    movel([0.108548, -1.229581, -2.664379, -0.818429, 1.570796, 1.679344],accel_mss,speed_ms,0,blend_radius_m)
    movel([0.107464, -1.232991, -2.662638, -0.816759, 1.570796, 1.678260],accel_mss,speed_ms,0,blend_radius_m)
    movel([0.106659, -1.236345, -2.660913, -0.815131, 1.570796, 1.677455],accel_mss,speed_ms,0,blend_radius_m)
    movel([0.106148, -1.239625, -2.659213, -0.813551, 1.570796, 1.676944],accel_mss,speed_ms,0,blend_radius_m)
    movel([0.105928, -1.242820, -2.657545, -0.812024, 1.570796, 1.676724],accel_mss,speed_ms,0,blend_radius_m)
    movel([0.106013, -1.245914, -2.655918, -0.810557, 1.570796, 1.676809],accel_mss,speed_ms,0,blend_radius_m)
    movel([0.106368, -1.248628, -2.654481, -0.809280, 1.570796, 1.677165],accel_mss,speed_ms,0,blend_radius_m)
    movel([0.106979, -1.251120, -2.653154, -0.808115, 1.570796, 1.677775],accel_mss,speed_ms,0,blend_radius_m)
    movel([0.107817, -1.253397, -2.651935, -0.807057, 1.570796, 1.678614],accel_mss,speed_ms,0,blend_radius_m)
    movel([0.108863, -1.255463, -2.650824, -0.806102, 1.570796, 1.679659],accel_mss,speed_ms,0,blend_radius_m)
    movel([0.110091, -1.257325, -2.649818, -0.805246, 1.570796, 1.680887],accel_mss,speed_ms,0,blend_radius_m)
    movel([0.111476, -1.258987, -2.648916, -0.804485, 1.570796, 1.682272],accel_mss,speed_ms,0,blend_radius_m)
    movel([0.112995, -1.260456, -2.648117, -0.803816, 1.570796, 1.683792],accel_mss,speed_ms,0,blend_radius_m)
    movel([0.114629, -1.261734, -2.647419, -0.803236, 1.570796, 1.685426],accel_mss,speed_ms,0,blend_radius_m)
    movel([0.116356, -1.262825, -2.646822, -0.802742, 1.570796, 1.687152],accel_mss,speed_ms,0,blend_radius_m)
    movel([0.118150, -1.263736, -2.646322, -0.802331, 1.570796, 1.688947],accel_mss,speed_ms,0,blend_radius_m)
    movel([0.119994, -1.264467, -2.645920, -0.802002, 1.570796, 1.690791],accel_mss,speed_ms,0,blend_radius_m)
    movel([0.121863, -1.265023, -2.645614, -0.801752, 1.570796, 1.692659],accel_mss,speed_ms,0,blend_radius_m)
    movel([0.123738, -1.265404, -2.645404, -0.801581, 1.570796, 1.694534],accel_mss,speed_ms,0,blend_radius_m)
    movel([0.125599, -1.265611, -2.645290, -0.801488, 1.570796, 1.696395],accel_mss,speed_ms,0,blend_radius_m)
    movel([0.127421, -1.265653, -2.645267, -0.801469, 1.570796, 1.698217],accel_mss,speed_ms,0,blend_radius_m)
    movel([0.129187, -1.265524, -2.645338, -0.801527, 1.570796, 1.699983],accel_mss,speed_ms,0,blend_radius_m)
    movel([0.130799, -1.262042, -2.647250, -0.803096, 1.570796, 1.701596],accel_mss,speed_ms,0,blend_radius_m)
    movel([0.127034, -1.261584, -2.647501, -0.803304, 1.570796, 1.697831],accel_mss,speed_ms,0,blend_radius_m)
    movel([0.123670, -1.260748, -2.647958, -0.803684, 1.570796, 1.694467],accel_mss,speed_ms,0,blend_radius_m)
    movel([0.120699, -1.259562, -2.648603, -0.804223, 1.570796, 1.691495],accel_mss,speed_ms,0,blend_radius_m)
    movel([0.118110, -1.258051, -2.649424, -0.804913, 1.570796, 1.688906],accel_mss,speed_ms,0,blend_radius_m)
    movel([0.115901, -1.256233, -2.650408, -0.805748, 1.570796, 1.686697],accel_mss,speed_ms,0,blend_radius_m)
    movel([0.114064, -1.254135, -2.651539, -0.806715, 1.570796, 1.684861],accel_mss,speed_ms,0,blend_radius_m)
    movel([0.112599, -1.251775, -2.652804, -0.807810, 1.570796, 1.683395],accel_mss,speed_ms,0,blend_radius_m)
    movel([0.111497, -1.249180, -2.654188, -0.809021, 1.570796, 1.682294],accel_mss,speed_ms,0,blend_radius_m)
    movel([0.110757, -1.246371, -2.655676, -0.810342, 1.570796, 1.681553],accel_mss,speed_ms,0,blend_radius_m)
    movel([0.110373, -1.243371, -2.657256, -0.811762, 1.570796, 1.681169],accel_mss,speed_ms,0,blend_radius_m)
    movel([0.110346, -1.240205, -2.658911, -0.813273, 1.570796, 1.681143],accel_mss,speed_ms,0,blend_radius_m)
    movel([0.110668, -1.236899, -2.660627, -0.814863, 1.570796, 1.681464],accel_mss,speed_ms,0,blend_radius_m)
    movel([0.111341, -1.233474, -2.662391, -0.816524, 1.570796, 1.682137],accel_mss,speed_ms,0,blend_radius_m)
    movel([0.112362, -1.229961, -2.664186, -0.818242, 1.570796, 1.683158],accel_mss,speed_ms,0,blend_radius_m)
    movel([0.113724, -1.226382, -2.666000, -0.820007, 1.570796, 1.684520],accel_mss,speed_ms,0,blend_radius_m)
    movel([0.115426, -1.222769, -2.667817, -0.821803, 1.570796, 1.686223],accel_mss,speed_ms,0,blend_radius_m)
    movel([0.117544, -1.218987, -2.669702, -0.823699, 1.570796, 1.688341],accel_mss,speed_ms,0,blend_radius_m)
    movel([0.119932, -1.215305, -2.671523, -0.825562, 1.570796, 1.690729],accel_mss,speed_ms,0,blend_radius_m)
    movel([0.122570, -1.211733, -2.673273, -0.827383, 1.570796, 1.693366],accel_mss,speed_ms,0,blend_radius_m)
    movel([0.125434, -1.208299, -2.674943, -0.829147, 1.570796, 1.696231],accel_mss,speed_ms,0,blend_radius_m)
    movel([0.128500, -1.205022, -2.676524, -0.830843, 1.570796, 1.699296],accel_mss,speed_ms,0,blend_radius_m)
    movel([0.131747, -1.201919, -2.678010, -0.832459, 1.570796, 1.702544],accel_mss,speed_ms,0,blend_radius_m)
    movel([0.135148, -1.199015, -2.679392, -0.833982, 1.570796, 1.705945],accel_mss,speed_ms,0,blend_radius_m)
    movel([0.138679, -1.196328, -2.680662, -0.835399, 1.570796, 1.709475],accel_mss,speed_ms,0,blend_radius_m)
    movel([0.142314, -1.193882, -2.681811, -0.836696, 1.570796, 1.713110],accel_mss,speed_ms,0,blend_radius_m)
    movel([0.146026, -1.191698, -2.682831, -0.837859, 1.570796, 1.716822],accel_mss,speed_ms,0,blend_radius_m)
    movel([0.149789, -1.189798, -2.683715, -0.838876, 1.570796, 1.720586],accel_mss,speed_ms,0,blend_radius_m)
    movel([0.153576, -1.188205, -2.684453, -0.839731, 1.570796, 1.724373],accel_mss,speed_ms,0,blend_radius_m)
    movel([0.157357, -1.186934, -2.685039, -0.840415, 1.570796, 1.728154],accel_mss,speed_ms,0,blend_radius_m)
    movel([0.161105, -1.186010, -2.685465, -0.840914, 1.570796, 1.731901],accel_mss,speed_ms,0,blend_radius_m)
    movel([0.164790, -1.185454, -2.685721, -0.841214, 1.570796, 1.735586],accel_mss,speed_ms,0,blend_radius_m)
    movel([0.168388, -1.185281, -2.685800, -0.841308, 1.570796, 1.739184],accel_mss,speed_ms,0,blend_radius_m)
    movel([0.171744, -1.185486, -2.685706, -0.841197, 1.570796, 1.742541],accel_mss,speed_ms,0,blend_radius_m)
    movel([0.174813, -1.186046, -2.685449, -0.840895, 1.570796, 1.745609],accel_mss,speed_ms,0,blend_radius_m)
    movel([0.177595, -1.186957, -2.685029, -0.840403, 1.570796, 1.748391],accel_mss,speed_ms,0,blend_radius_m)
    movel([0.180079, -1.188212, -2.684450, -0.839728, 1.570796, 1.750875],accel_mss,speed_ms,0,blend_radius_m)
    movel([0.182267, -1.189808, -2.683710, -0.838870, 1.570796, 1.753063],accel_mss,speed_ms,0,blend_radius_m)
    movel([0.184151, -1.191740, -2.682812, -0.837837, 1.570796, 1.754947],accel_mss,speed_ms,0,blend_radius_m)
    movel([0.185731, -1.194002, -2.681755, -0.836632, 1.570796, 1.756527],accel_mss,speed_ms,0,blend_radius_m)
    movel([0.187008, -1.196584, -2.680541, -0.835264, 1.570796, 1.757804],accel_mss,speed_ms,0,blend_radius_m)
    movel([0.188195, -1.200365, -2.678751, -0.833273, 1.570796, 1.758991],accel_mss,speed_ms,0,blend_radius_m)
    movel([0.188551, -1.202327, -2.677816, -0.832246, 1.570796, 1.759347],accel_mss,speed_ms,0,blend_radius_m)
    movel([0.188803, -1.206387, -2.675867, -0.830135, 1.570796, 1.759599],accel_mss,speed_ms,0,blend_radius_m)
    movel([0.188703, -1.208484, -2.674853, -0.829051, 1.570796, 1.759500],accel_mss,speed_ms,0,blend_radius_m)
    movel([0.188070, -1.212794, -2.672754, -0.826840, 1.570796, 1.758866],accel_mss,speed_ms,0,blend_radius_m)
    movel([0.187544, -1.215004, -2.671670, -0.825715, 1.570796, 1.758341],accel_mss,speed_ms,0,blend_radius_m)
    movel([0.186076, -1.219536, -2.669430, -0.823423, 1.570796, 1.756872],accel_mss,speed_ms,0,blend_radius_m)
    movel([0.185142, -1.221849, -2.668277, -0.822263, 1.570796, 1.755939],accel_mss,speed_ms,0,blend_radius_m)
    movel([0.182886, -1.226576, -2.665902, -0.819911, 1.570796, 1.753682],accel_mss,speed_ms,0,blend_radius_m)
    movel([0.180136, -1.231422, -2.663441, -0.817526, 1.570796, 1.750932],accel_mss,speed_ms,0,blend_radius_m)
    movel([0.183278, -1.232244, -2.663021, -0.817124, 1.570796, 1.754074],accel_mss,speed_ms,0,blend_radius_m)
    movel([0.185050, -1.229577, -2.664381, -0.818430, 1.570796, 1.755846],accel_mss,speed_ms,0,blend_radius_m)
    movel([0.185168, -1.229377, -2.664483, -0.818529, 1.570796, 1.755964],accel_mss,speed_ms,0,blend_radius_m)
    speed_ms = 0.005
    # Splitting Linear movement in 4 (instruction 1141: MoveL 1073)
    movel([0.185168, -1.226955, -2.663319, -0.822115, 1.570796, 1.755964],accel_mss,speed_ms,0,blend_radius_m)
    movel([0.185168, -1.224548, -2.662151, -0.825690, 1.570796, 1.755964],accel_mss,speed_ms,0,blend_radius_m)
    movel([0.185168, -1.222156, -2.660979, -0.829253, 1.570796, 1.755964],accel_mss,speed_ms,0,blend_radius_m)
    movel([0.185168, -1.219779, -2.659804, -0.832806, 1.570796, 1.755964],accel_mss,speed_ms,0,blend_radius_m)
    speed_ms = 0.040
    # Splitting Linear movement in 8 (instruction 1143: MoveL 1074)
    movel([0.184772, -1.222069, -2.658652, -0.831667, 1.570796, 1.755568],accel_mss,speed_ms,0,blend_radius_m)
    movel([0.184379, -1.224351, -2.657499, -0.830539, 1.570796, 1.755175],accel_mss,speed_ms,0,blend_radius_m)
    movel([0.183987, -1.226625, -2.656343, -0.829421, 1.570796, 1.754783],accel_mss,speed_ms,0,blend_radius_m)
    movel([0.183597, -1.228891, -2.655186, -0.828312, 1.570796, 1.754394],accel_mss,speed_ms,0,blend_radius_m)
    movel([0.183210, -1.231149, -2.654027, -0.827213, 1.570796, 1.754006],accel_mss,speed_ms,0,blend_radius_m)
    movel([0.182824, -1.233399, -2.652866, -0.826124, 1.570796, 1.753620],accel_mss,speed_ms,0,blend_radius_m)
    movel([0.182440, -1.235641, -2.651703, -0.825045, 1.570796, 1.753237],accel_mss,speed_ms,0,blend_radius_m)
    movel([0.182059, -1.237876, -2.650538, -0.823975, 1.570796, 1.752855],accel_mss,speed_ms,0,blend_radius_m)
    speed_ms = 0.005
    # Splitting Linear movement in 4 (instruction 1145: MoveL 1075)
    movel([0.182059, -1.240234, -2.651693, -0.820462, 1.570796, 1.752855],accel_mss,speed_ms,0,blend_radius_m)
    movel([0.182059, -1.242607, -2.652844, -0.816938, 1.570796, 1.752855],accel_mss,speed_ms,0,blend_radius_m)
    movel([0.182059, -1.244994, -2.653991, -0.813404, 1.570796, 1.752855],accel_mss,speed_ms,0,blend_radius_m)
    movel([0.182059, -1.247395, -2.655135, -0.809860, 1.570796, 1.752855],accel_mss,speed_ms,0,blend_radius_m)
    speed_ms = 0.035
    movel([0.183122, -1.249001, -2.654283, -0.809105, 1.570796, 1.753919],accel_mss,speed_ms,0,blend_radius_m)
    movel([0.184641, -1.250273, -2.653606, -0.808510, 1.570796, 1.755437],accel_mss,speed_ms,0,blend_radius_m)
    movel([0.186541, -1.251208, -2.653107, -0.808074, 1.570796, 1.757337],accel_mss,speed_ms,0,blend_radius_m)
    movel([0.188759, -1.251797, -2.652792, -0.807799, 1.570796, 1.759556],accel_mss,speed_ms,0,blend_radius_m)
    movel([0.191228, -1.252032, -2.652667, -0.807690, 1.570796, 1.762025],accel_mss,speed_ms,0,blend_radius_m)
    movel([0.193881, -1.251908, -2.652733, -0.807748, 1.570796, 1.764677],accel_mss,speed_ms,0,blend_radius_m)
    movel([0.196654, -1.251410, -2.652999, -0.807980, 1.570796, 1.767451],accel_mss,speed_ms,0,blend_radius_m)
    movel([0.199484, -1.250525, -2.653471, -0.808392, 1.570796, 1.770280],accel_mss,speed_ms,0,blend_radius_m)
    movel([0.202221, -1.249329, -2.654109, -0.808952, 1.570796, 1.773017],accel_mss,speed_ms,0,blend_radius_m)
    movel([0.204953, -1.247840, -2.654899, -0.809650, 1.570796, 1.775749],accel_mss,speed_ms,0,blend_radius_m)
    movel([0.207603, -1.246119, -2.655809, -0.810461, 1.570796, 1.778399],accel_mss,speed_ms,0,blend_radius_m)
    movel([0.210103, -1.244221, -2.656809, -0.811359, 1.570796, 1.780900],accel_mss,speed_ms,0,blend_radius_m)
    movel([0.212379, -1.242201, -2.657869, -0.812319, 1.570796, 1.783175],accel_mss,speed_ms,0,blend_radius_m)
    movel([0.214355, -1.240118, -2.658956, -0.813315, 1.570796, 1.785152],accel_mss,speed_ms,0,blend_radius_m)
    movel([0.215949, -1.238033, -2.660040, -0.814316, 1.570796, 1.786746],accel_mss,speed_ms,0,blend_radius_m)
    movel([0.217091, -1.236001, -2.661090, -0.815297, 1.570796, 1.787887],accel_mss,speed_ms,0,blend_radius_m)
    movel([0.214017, -1.235343, -2.661430, -0.815616, 1.570796, 1.784814],accel_mss,speed_ms,0,blend_radius_m)
    movel([0.212357, -1.237457, -2.660338, -0.814594, 1.570796, 1.783154],accel_mss,speed_ms,0,blend_radius_m)
    movel([0.210630, -1.239382, -2.659339, -0.813668, 1.570796, 1.781426],accel_mss,speed_ms,0,blend_radius_m)
    movel([0.208832, -1.241125, -2.658431, -0.812833, 1.570796, 1.779628],accel_mss,speed_ms,0,blend_radius_m)
    movel([0.206964, -1.242679, -2.657619, -0.812092, 1.570796, 1.777760],accel_mss,speed_ms,0,blend_radius_m)
    movel([0.205021, -1.244043, -2.656903, -0.811443, 1.570796, 1.775817],accel_mss,speed_ms,0,blend_radius_m)
    movel([0.202999, -1.245224, -2.656281, -0.810884, 1.570796, 1.773795],accel_mss,speed_ms,0,blend_radius_m)
    movel([0.200896, -1.246213, -2.655760, -0.810416, 1.570796, 1.771693],accel_mss,speed_ms,0,blend_radius_m)
    movel([0.198709, -1.247009, -2.655339, -0.810041, 1.570796, 1.769506],accel_mss,speed_ms,0,blend_radius_m)
    movel([0.196531, -1.247582, -2.655036, -0.809771, 1.570796, 1.767327],accel_mss,speed_ms,0,blend_radius_m)
    movel([0.194520, -1.247878, -2.654879, -0.809632, 1.570796, 1.765316],accel_mss,speed_ms,0,blend_radius_m)
    movel([0.192672, -1.247905, -2.654865, -0.809620, 1.570796, 1.763468],accel_mss,speed_ms,0,blend_radius_m)
    movel([0.190982, -1.247672, -2.654988, -0.809729, 1.570796, 1.761779],accel_mss,speed_ms,0,blend_radius_m)
    movel([0.189441, -1.247187, -2.655245, -0.809957, 1.570796, 1.760237],accel_mss,speed_ms,0,blend_radius_m)
    movel([0.188048, -1.246455, -2.655632, -0.810302, 1.570796, 1.758845],accel_mss,speed_ms,0,blend_radius_m)
    movel([0.186797, -1.245483, -2.656145, -0.810761, 1.570796, 1.757594],accel_mss,speed_ms,0,blend_radius_m)
    movel([0.185682, -1.244282, -2.656777, -0.811330, 1.570796, 1.756478],accel_mss,speed_ms,0,blend_radius_m)
    movel([0.182059, -1.247395, -2.655135, -0.809860, 1.570796, 1.752855],accel_mss,speed_ms,0,blend_radius_m)
    movel([0.183122, -1.249001, -2.654283, -0.809105, 1.570796, 1.753919],accel_mss,speed_ms,0,blend_radius_m)
    movel([0.183292, -1.249140, -2.654209, -0.809040, 1.570796, 1.754088],accel_mss,speed_ms,0,blend_radius_m)
    speed_ms = 0.005
    # Splitting Linear movement in 6 (instruction 1184: MoveL 1112)
    movel([0.183292, -1.247540, -2.653448, -0.811401, 1.570796, 1.754088],accel_mss,speed_ms,0,blend_radius_m)
    movel([0.183292, -1.245945, -2.652686, -0.813758, 1.570796, 1.754088],accel_mss,speed_ms,0,blend_radius_m)
    movel([0.183292, -1.244357, -2.651922, -0.816110, 1.570796, 1.754088],accel_mss,speed_ms,0,blend_radius_m)
    movel([0.183292, -1.242775, -2.651156, -0.818458, 1.570796, 1.754088],accel_mss,speed_ms,0,blend_radius_m)
    movel([0.183292, -1.241199, -2.650389, -0.820801, 1.570796, 1.754088],accel_mss,speed_ms,0,blend_radius_m)
    movel([0.183292, -1.239630, -2.649620, -0.823139, 1.570796, 1.754088],accel_mss,speed_ms,0,blend_radius_m)
    speed_ms = 0.040
    # Splitting Linear movement in 18 (instruction 1186: MoveL 1113)
    movel([0.186032, -1.238792, -2.650059, -0.823538, 1.570796, 1.756828],accel_mss,speed_ms,0,blend_radius_m)
    movel([0.188773, -1.237959, -2.650495, -0.823935, 1.570796, 1.759569],accel_mss,speed_ms,0,blend_radius_m)
    movel([0.191516, -1.237130, -2.650927, -0.824331, 1.570796, 1.762312],accel_mss,speed_ms,0,blend_radius_m)
    movel([0.194260, -1.236307, -2.651357, -0.824726, 1.570796, 1.765056],accel_mss,speed_ms,0,blend_radius_m)
    movel([0.197005, -1.235488, -2.651782, -0.825118, 1.570796, 1.767802],accel_mss,speed_ms,0,blend_radius_m)
    movel([0.199752, -1.234675, -2.652205, -0.825509, 1.570796, 1.770548],accel_mss,speed_ms,0,blend_radius_m)
    movel([0.202500, -1.233866, -2.652624, -0.825899, 1.570796, 1.773297],accel_mss,speed_ms,0,blend_radius_m)
    movel([0.205250, -1.233063, -2.653039, -0.826287, 1.570796, 1.776046],accel_mss,speed_ms,0,blend_radius_m)
    movel([0.208000, -1.232265, -2.653452, -0.826673, 1.570796, 1.778796],accel_mss,speed_ms,0,blend_radius_m)
    movel([0.210752, -1.231471, -2.653861, -0.827057, 1.570796, 1.781548],accel_mss,speed_ms,0,blend_radius_m)
    movel([0.213505, -1.230683, -2.654266, -0.827440, 1.570796, 1.784301],accel_mss,speed_ms,0,blend_radius_m)
    movel([0.216259, -1.229900, -2.654668, -0.827820, 1.570796, 1.787055],accel_mss,speed_ms,0,blend_radius_m)
    movel([0.219014, -1.229122, -2.655067, -0.828199, 1.570796, 1.789810],accel_mss,speed_ms,0,blend_radius_m)
    movel([0.221770, -1.228350, -2.655463, -0.828576, 1.570796, 1.792566],accel_mss,speed_ms,0,blend_radius_m)
    movel([0.224526, -1.227583, -2.655855, -0.828951, 1.570796, 1.795323],accel_mss,speed_ms,0,blend_radius_m)
    movel([0.227284, -1.226821, -2.656243, -0.829325, 1.570796, 1.798081],accel_mss,speed_ms,0,blend_radius_m)
    movel([0.230043, -1.226064, -2.656629, -0.829696, 1.570796, 1.800839],accel_mss,speed_ms,0,blend_radius_m)
    movel([0.232803, -1.225313, -2.657011, -0.830065, 1.570796, 1.803599],accel_mss,speed_ms,0,blend_radius_m)
    speed_ms = 0.005
    # Splitting Linear movement in 6 (instruction 1188: MoveL 1114)
    movel([0.232803, -1.226893, -2.657790, -0.827706, 1.570796, 1.803599],accel_mss,speed_ms,0,blend_radius_m)
    movel([0.232803, -1.228479, -2.658568, -0.825342, 1.570796, 1.803599],accel_mss,speed_ms,0,blend_radius_m)
    movel([0.232803, -1.230072, -2.659345, -0.822973, 1.570796, 1.803599],accel_mss,speed_ms,0,blend_radius_m)
    movel([0.232803, -1.231670, -2.660119, -0.820599, 1.570796, 1.803599],accel_mss,speed_ms,0,blend_radius_m)
    movel([0.232803, -1.233276, -2.660893, -0.818220, 1.570796, 1.803599],accel_mss,speed_ms,0,blend_radius_m)
    movel([0.232803, -1.234888, -2.661664, -0.815837, 1.570796, 1.803599],accel_mss,speed_ms,0,blend_radius_m)
    speed_ms = 0.035
    movel([0.230920, -1.234418, -2.661906, -0.816065, 1.570796, 1.801717],accel_mss,speed_ms,0,blend_radius_m)
    movel([0.230264, -1.234390, -2.661921, -0.816079, 1.570796, 1.801060],accel_mss,speed_ms,0,blend_radius_m)
    movel([0.229709, -1.234540, -2.661843, -0.816006, 1.570796, 1.800506],accel_mss,speed_ms,0,blend_radius_m)
    movel([0.229199, -1.234894, -2.661661, -0.815834, 1.570796, 1.799995],accel_mss,speed_ms,0,blend_radius_m)
    movel([0.228657, -1.235491, -2.661354, -0.815544, 1.570796, 1.799454],accel_mss,speed_ms,0,blend_radius_m)
    movel([0.225246, -1.240320, -2.658851, -0.813218, 1.570796, 1.796042],accel_mss,speed_ms,0,blend_radius_m)
    movel([0.223109, -1.242993, -2.657454, -0.811942, 1.570796, 1.793906],accel_mss,speed_ms,0,blend_radius_m)
    movel([0.220844, -1.245530, -2.656120, -0.810739, 1.570796, 1.791641],accel_mss,speed_ms,0,blend_radius_m)
    movel([0.218468, -1.247920, -2.654856, -0.809612, 1.570796, 1.789264],accel_mss,speed_ms,0,blend_radius_m)
    movel([0.215996, -1.250161, -2.653665, -0.808562, 1.570796, 1.786792],accel_mss,speed_ms,0,blend_radius_m)
    movel([0.213445, -1.252238, -2.652556, -0.807594, 1.570796, 1.784242],accel_mss,speed_ms,0,blend_radius_m)
    movel([0.210829, -1.254150, -2.651531, -0.806708, 1.570796, 1.781626],accel_mss,speed_ms,0,blend_radius_m)
    movel([0.208160, -1.255889, -2.650594, -0.805906, 1.570796, 1.778956],accel_mss,speed_ms,0,blend_radius_m)
    movel([0.205457, -1.257445, -2.649753, -0.805191, 1.570796, 1.776253],accel_mss,speed_ms,0,blend_radius_m)
    movel([0.202731, -1.258811, -2.649012, -0.804566, 1.570796, 1.773527],accel_mss,speed_ms,0,blend_radius_m)
    movel([0.200000, -1.259978, -2.648377, -0.804034, 1.570796, 1.770796],accel_mss,speed_ms,0,blend_radius_m)
    movel([0.197273, -1.260941, -2.647852, -0.803596, 1.570796, 1.768070],accel_mss,speed_ms,0,blend_radius_m)
    movel([0.194565, -1.261691, -2.647442, -0.803256, 1.570796, 1.765361],accel_mss,speed_ms,0,blend_radius_m)
    movel([0.191894, -1.262218, -2.647154, -0.803017, 1.570796, 1.762691],accel_mss,speed_ms,0,blend_radius_m)
    movel([0.189269, -1.262516, -2.646991, -0.802882, 1.570796, 1.760065],accel_mss,speed_ms,0,blend_radius_m)
    movel([0.186708, -1.262571, -2.646961, -0.802857, 1.570796, 1.757504],accel_mss,speed_ms,0,blend_radius_m)
    movel([0.183681, -1.262322, -2.647097, -0.802970, 1.570796, 1.754477],accel_mss,speed_ms,0,blend_radius_m)
    movel([0.180930, -1.261741, -2.647415, -0.803233, 1.570796, 1.751727],accel_mss,speed_ms,0,blend_radius_m)
    movel([0.178461, -1.260852, -2.647901, -0.803636, 1.570796, 1.749257],accel_mss,speed_ms,0,blend_radius_m)
    movel([0.176271, -1.259665, -2.648547, -0.804176, 1.570796, 1.747068],accel_mss,speed_ms,0,blend_radius_m)
    movel([0.174378, -1.258199, -2.649344, -0.804846, 1.570796, 1.745174],accel_mss,speed_ms,0,blend_radius_m)
    movel([0.172780, -1.256464, -2.650284, -0.805642, 1.570796, 1.743576],accel_mss,speed_ms,0,blend_radius_m)
    movel([0.171488, -1.254480, -2.651353, -0.806556, 1.570796, 1.742284],accel_mss,speed_ms,0,blend_radius_m)
    movel([0.170509, -1.252257, -2.652546, -0.807586, 1.570796, 1.741305],accel_mss,speed_ms,0,blend_radius_m)
    movel([0.169853, -1.249811, -2.653852, -0.808726, 1.570796, 1.740650],accel_mss,speed_ms,0,blend_radius_m)
    movel([0.169531, -1.247155, -2.655262, -0.809972, 1.570796, 1.740327],accel_mss,speed_ms,0,blend_radius_m)
    movel([0.169549, -1.244305, -2.656765, -0.811319, 1.570796, 1.740346],accel_mss,speed_ms,0,blend_radius_m)
    movel([0.169920, -1.241274, -2.658353, -0.812762, 1.570796, 1.740717],accel_mss,speed_ms,0,blend_radius_m)
    movel([0.170655, -1.238077, -2.660017, -0.814295, 1.570796, 1.741451],accel_mss,speed_ms,0,blend_radius_m)
    movel([0.171759, -1.234730, -2.661746, -0.815914, 1.570796, 1.742556],accel_mss,speed_ms,0,blend_radius_m)
    movel([0.173248, -1.231249, -2.663530, -0.817611, 1.570796, 1.744045],accel_mss,speed_ms,0,blend_radius_m)
    movel([0.175135, -1.227646, -2.665361, -0.819382, 1.570796, 1.745931],accel_mss,speed_ms,0,blend_radius_m)
    movel([0.175741, -1.226245, -2.666070, -0.820075, 1.570796, 1.746537],accel_mss,speed_ms,0,blend_radius_m)
    movel([0.175768, -1.225786, -2.666301, -0.820302, 1.570796, 1.746565],accel_mss,speed_ms,0,blend_radius_m)
    movel([0.175649, -1.225448, -2.666471, -0.820470, 1.570796, 1.746445],accel_mss,speed_ms,0,blend_radius_m)
    movel([0.175056, -1.225044, -2.666675, -0.820670, 1.570796, 1.745852],accel_mss,speed_ms,0,blend_radius_m)
    movel([0.173610, -1.224769, -2.666813, -0.820807, 1.570796, 1.744407],accel_mss,speed_ms,0,blend_radius_m)
    movel([0.173153, -1.224865, -2.666765, -0.820759, 1.570796, 1.743950],accel_mss,speed_ms,0,blend_radius_m)
    movel([0.172770, -1.225077, -2.666658, -0.820654, 1.570796, 1.743567],accel_mss,speed_ms,0,blend_radius_m)
    movel([0.172444, -1.225380, -2.666505, -0.820503, 1.570796, 1.743240],accel_mss,speed_ms,0,blend_radius_m)
    movel([0.171457, -1.226980, -2.665698, -0.819711, 1.570796, 1.742253],accel_mss,speed_ms,0,blend_radius_m)
    movel([0.170206, -1.229224, -2.664561, -0.818604, 1.570796, 1.741002],accel_mss,speed_ms,0,blend_radius_m)
    movel([0.168132, -1.233602, -2.662325, -0.816462, 1.570796, 1.738928],accel_mss,speed_ms,0,blend_radius_m)
    movel([0.167304, -1.235729, -2.661231, -0.815429, 1.570796, 1.738100],accel_mss,speed_ms,0,blend_radius_m)
    movel([0.166050, -1.239846, -2.659098, -0.813445, 1.570796, 1.736847],accel_mss,speed_ms,0,blend_radius_m)
    movel([0.165319, -1.243754, -2.657054, -0.811580, 1.570796, 1.736116],accel_mss,speed_ms,0,blend_radius_m)
    movel([0.165086, -1.247433, -2.655115, -0.809842, 1.570796, 1.735882],accel_mss,speed_ms,0,blend_radius_m)
    movel([0.165329, -1.250861, -2.653292, -0.808236, 1.570796, 1.736125],accel_mss,speed_ms,0,blend_radius_m)
    movel([0.166030, -1.254012, -2.651605, -0.806772, 1.570796, 1.736827],accel_mss,speed_ms,0,blend_radius_m)
    movel([0.167168, -1.256866, -2.650066, -0.805457, 1.570796, 1.737964],accel_mss,speed_ms,0,blend_radius_m)
    movel([0.168727, -1.259401, -2.648691, -0.804297, 1.570796, 1.739523],accel_mss,speed_ms,0,blend_radius_m)
    movel([0.170690, -1.261594, -2.647495, -0.803300, 1.570796, 1.741486],accel_mss,speed_ms,0,blend_radius_m)
    movel([0.173040, -1.263420, -2.646495, -0.802474, 1.570796, 1.743836],accel_mss,speed_ms,0,blend_radius_m)
    movel([0.175759, -1.264863, -2.645702, -0.801824, 1.570796, 1.746555],accel_mss,speed_ms,0,blend_radius_m)
    movel([0.178840, -1.265892, -2.645135, -0.801362, 1.570796, 1.749636],accel_mss,speed_ms,0,blend_radius_m)
    movel([0.180510, -1.266245, -2.644940, -0.801204, 1.570796, 1.751306],accel_mss,speed_ms,0,blend_radius_m)
    movel([0.184106, -1.266610, -2.644738, -0.801041, 1.570796, 1.754902],accel_mss,speed_ms,0,blend_radius_m)
    movel([0.186028, -1.266617, -2.644735, -0.801038, 1.570796, 1.756825],accel_mss,speed_ms,0,blend_radius_m)
    movel([0.190118, -1.266257, -2.644933, -0.801199, 1.570796, 1.760914],accel_mss,speed_ms,0,blend_radius_m)
    movel([0.191256, -1.266232, -2.644947, -0.801210, 1.570796, 1.762052],accel_mss,speed_ms,0,blend_radius_m)
    movel([0.191977, -1.266551, -2.644771, -0.801067, 1.570796, 1.762774],accel_mss,speed_ms,0,blend_radius_m)
    movel([0.192328, -1.267205, -2.644409, -0.800775, 1.570796, 1.763125],accel_mss,speed_ms,0,blend_radius_m)
    movel([0.192350, -1.268195, -2.643860, -0.800333, 1.570796, 1.763146],accel_mss,speed_ms,0,blend_radius_m)
    movel([0.192192, -1.269028, -2.643398, -0.799963, 1.570796, 1.762989],accel_mss,speed_ms,0,blend_radius_m)
    movel([0.191509, -1.270658, -2.642491, -0.799241, 1.570796, 1.762306],accel_mss,speed_ms,0,blend_radius_m)
    movel([0.190999, -1.271435, -2.642057, -0.798897, 1.570796, 1.761795],accel_mss,speed_ms,0,blend_radius_m)
    movel([0.189676, -1.272866, -2.641256, -0.798267, 1.570796, 1.760472],accel_mss,speed_ms,0,blend_radius_m)
    movel([0.188880, -1.273500, -2.640900, -0.797989, 1.570796, 1.759676],accel_mss,speed_ms,0,blend_radius_m)
    movel([0.187157, -1.274501, -2.640338, -0.797550, 1.570796, 1.757953],accel_mss,speed_ms,0,blend_radius_m)
    movel([0.186313, -1.274824, -2.640156, -0.797409, 1.570796, 1.757109],accel_mss,speed_ms,0,blend_radius_m)
    movel([0.184714, -1.275107, -2.639996, -0.797285, 1.570796, 1.755510],accel_mss,speed_ms,0,blend_radius_m)
    movel([0.184004, -1.275055, -2.640026, -0.797308, 1.570796, 1.754800],accel_mss,speed_ms,0,blend_radius_m)
    movel([0.183383, -1.274862, -2.640135, -0.797392, 1.570796, 1.754179],accel_mss,speed_ms,0,blend_radius_m)
    movel([0.182873, -1.274520, -2.640327, -0.797542, 1.570796, 1.753670],accel_mss,speed_ms,0,blend_radius_m)
    movel([0.182496, -1.274022, -2.640607, -0.797760, 1.570796, 1.753292],accel_mss,speed_ms,0,blend_radius_m)
    movel([0.182072, -1.273430, -2.640940, -0.798019, 1.570796, 1.752869],accel_mss,speed_ms,0,blend_radius_m)
    movel([0.181586, -1.273127, -2.641110, -0.798153, 1.570796, 1.752382],accel_mss,speed_ms,0,blend_radius_m)
    movel([0.181046, -1.273063, -2.641145, -0.798180, 1.570796, 1.751843],accel_mss,speed_ms,0,blend_radius_m)
    movel([0.180458, -1.273194, -2.641072, -0.798123, 1.570796, 1.751254],accel_mss,speed_ms,0,blend_radius_m)
    movel([0.179180, -1.273838, -2.640710, -0.797840, 1.570796, 1.749976],accel_mss,speed_ms,0,blend_radius_m)
    movel([0.177812, -1.274672, -2.640242, -0.797475, 1.570796, 1.748609],accel_mss,speed_ms,0,blend_radius_m)
    movel([0.178144, -1.276063, -2.639458, -0.796869, 1.570796, 1.748940],accel_mss,speed_ms,0,blend_radius_m)
    movel([0.178747, -1.277198, -2.638816, -0.796375, 1.570796, 1.749544],accel_mss,speed_ms,0,blend_radius_m)
    movel([0.179596, -1.278073, -2.638320, -0.795996, 1.570796, 1.750392],accel_mss,speed_ms,0,blend_radius_m)
    movel([0.180671, -1.278679, -2.637977, -0.795733, 1.570796, 1.751467],accel_mss,speed_ms,0,blend_radius_m)
    movel([0.181946, -1.279009, -2.637789, -0.795591, 1.570796, 1.752743],accel_mss,speed_ms,0,blend_radius_m)
    movel([0.183398, -1.279061, -2.637760, -0.795568, 1.570796, 1.754195],accel_mss,speed_ms,0,blend_radius_m)
    movel([0.185006, -1.278823, -2.637895, -0.795671, 1.570796, 1.755802],accel_mss,speed_ms,0,blend_radius_m)
    movel([0.186748, -1.278287, -2.638199, -0.795903, 1.570796, 1.757544],accel_mss,speed_ms,0,blend_radius_m)
    movel([0.188676, -1.277419, -2.638691, -0.796279, 1.570796, 1.759472],accel_mss,speed_ms,0,blend_radius_m)
    movel([0.190397, -1.276345, -2.639299, -0.796746, 1.570796, 1.761194],accel_mss,speed_ms,0,blend_radius_m)
    movel([0.191925, -1.275053, -2.640027, -0.797309, 1.570796, 1.762722],accel_mss,speed_ms,0,blend_radius_m)
    movel([0.193267, -1.273525, -2.640886, -0.797978, 1.570796, 1.764063],accel_mss,speed_ms,0,blend_radius_m)
    movel([0.194432, -1.271750, -2.641881, -0.798758, 1.570796, 1.765228],accel_mss,speed_ms,0,blend_radius_m)
    movel([0.195428, -1.269707, -2.643021, -0.799662, 1.570796, 1.766224],accel_mss,speed_ms,0,blend_radius_m)
    movel([0.196267, -1.267385, -2.644309, -0.800694, 1.570796, 1.767063],accel_mss,speed_ms,0,blend_radius_m)
    movel([0.196954, -1.264766, -2.645756, -0.801868, 1.570796, 1.767750],accel_mss,speed_ms,0,blend_radius_m)
    # Splitting Linear movement in 4 (instruction 1292: MoveL 1217)
    movel([0.198451, -1.264198, -2.646068, -0.802123, 1.570796, 1.769247],accel_mss,speed_ms,0,blend_radius_m)
    movel([0.199949, -1.263631, -2.646379, -0.802379, 1.570796, 1.770745],accel_mss,speed_ms,0,blend_radius_m)
    movel([0.201447, -1.263065, -2.646690, -0.802634, 1.570796, 1.772244],accel_mss,speed_ms,0,blend_radius_m)
    movel([0.202947, -1.262501, -2.646999, -0.802889, 1.570796, 1.773743],accel_mss,speed_ms,0,blend_radius_m)
    # Splitting Linear movement in 4 (instruction 1293: MoveL 1218)
    movel([0.203300, -1.263901, -2.646231, -0.802257, 1.570796, 1.774097],accel_mss,speed_ms,0,blend_radius_m)
    movel([0.203653, -1.265299, -2.645462, -0.801628, 1.570796, 1.774449],accel_mss,speed_ms,0,blend_radius_m)
    movel([0.204004, -1.266694, -2.644692, -0.801003, 1.570796, 1.774800],accel_mss,speed_ms,0,blend_radius_m)
    movel([0.204354, -1.268087, -2.643920, -0.800381, 1.570796, 1.775150],accel_mss,speed_ms,0,blend_radius_m)
    movel([0.204524, -1.268836, -2.643505, -0.800048, 1.570796, 1.775321],accel_mss,speed_ms,0,blend_radius_m)
    movel([0.204547, -1.269636, -2.643060, -0.799693, 1.570796, 1.775344],accel_mss,speed_ms,0,blend_radius_m)
    movel([0.204425, -1.270469, -2.642596, -0.799324, 1.570796, 1.775221],accel_mss,speed_ms,0,blend_radius_m)
    movel([0.204155, -1.271317, -2.642123, -0.798949, 1.570796, 1.774952],accel_mss,speed_ms,0,blend_radius_m)
    movel([0.203744, -1.272160, -2.641651, -0.798578, 1.570796, 1.774541],accel_mss,speed_ms,0,blend_radius_m)
    movel([0.203186, -1.272986, -2.641189, -0.798214, 1.570796, 1.773982],accel_mss,speed_ms,0,blend_radius_m)
    movel([0.202483, -1.273775, -2.640746, -0.797868, 1.570796, 1.773279],accel_mss,speed_ms,0,blend_radius_m)
    movel([0.201639, -1.274509, -2.640333, -0.797547, 1.570796, 1.772435],accel_mss,speed_ms,0,blend_radius_m)
    movel([0.200711, -1.275150, -2.639972, -0.797266, 1.570796, 1.771507],accel_mss,speed_ms,0,blend_radius_m)
    movel([0.199711, -1.275710, -2.639657, -0.797022, 1.570796, 1.770507],accel_mss,speed_ms,0,blend_radius_m)
    movel([0.198711, -1.276139, -2.639414, -0.796835, 1.570796, 1.769507],accel_mss,speed_ms,0,blend_radius_m)
    movel([0.197772, -1.276398, -2.639269, -0.796723, 1.570796, 1.768568],accel_mss,speed_ms,0,blend_radius_m)
    movel([0.197038, -1.276588, -2.639161, -0.796640, 1.570796, 1.767834],accel_mss,speed_ms,0,blend_radius_m)
    movel([0.196425, -1.276869, -2.639002, -0.796518, 1.570796, 1.767221],accel_mss,speed_ms,0,blend_radius_m)
    movel([0.195918, -1.277226, -2.638800, -0.796363, 1.570796, 1.766714],accel_mss,speed_ms,0,blend_radius_m)
    movel([0.195505, -1.277639, -2.638566, -0.796183, 1.570796, 1.766301],accel_mss,speed_ms,0,blend_radius_m)
    movel([0.194906, -1.278582, -2.638031, -0.795775, 1.570796, 1.765702],accel_mss,speed_ms,0,blend_radius_m)
    movel([0.194513, -1.279578, -2.637466, -0.795345, 1.570796, 1.765310],accel_mss,speed_ms,0,blend_radius_m)
    movel([0.194667, -1.279886, -2.637291, -0.795213, 1.570796, 1.765464],accel_mss,speed_ms,0,blend_radius_m)
    movel([0.195204, -1.280166, -2.637131, -0.795092, 1.570796, 1.766000],accel_mss,speed_ms,0,blend_radius_m)
    movel([0.195929, -1.280349, -2.637027, -0.795013, 1.570796, 1.766726],accel_mss,speed_ms,0,blend_radius_m)
    movel([0.196658, -1.280356, -2.637023, -0.795010, 1.570796, 1.767454],accel_mss,speed_ms,0,blend_radius_m)
    movel([0.198004, -1.280073, -2.637184, -0.795132, 1.570796, 1.768801],accel_mss,speed_ms,0,blend_radius_m)
    movel([0.199317, -1.279643, -2.637429, -0.795317, 1.570796, 1.770113],accel_mss,speed_ms,0,blend_radius_m)
    movel([0.200588, -1.279069, -2.637755, -0.795565, 1.570796, 1.771384],accel_mss,speed_ms,0,blend_radius_m)
    movel([0.201817, -1.278355, -2.638160, -0.795873, 1.570796, 1.772613],accel_mss,speed_ms,0,blend_radius_m)
    movel([0.202994, -1.277509, -2.638640, -0.796240, 1.570796, 1.773790],accel_mss,speed_ms,0,blend_radius_m)
    movel([0.204120, -1.276529, -2.639195, -0.796666, 1.570796, 1.774917],accel_mss,speed_ms,0,blend_radius_m)
    movel([0.205190, -1.275421, -2.639820, -0.797148, 1.570796, 1.775986],accel_mss,speed_ms,0,blend_radius_m)
    movel([0.206199, -1.274187, -2.640514, -0.797687, 1.570796, 1.776995],accel_mss,speed_ms,0,blend_radius_m)
    movel([0.207103, -1.272876, -2.641250, -0.798263, 1.570796, 1.777900],accel_mss,speed_ms,0,blend_radius_m)
    movel([0.207807, -1.271601, -2.641964, -0.798824, 1.570796, 1.778604],accel_mss,speed_ms,0,blend_radius_m)
    movel([0.208315, -1.270365, -2.642654, -0.799370, 1.570796, 1.779112],accel_mss,speed_ms,0,blend_radius_m)
    movel([0.208637, -1.269170, -2.643319, -0.799900, 1.570796, 1.779433],accel_mss,speed_ms,0,blend_radius_m)
    movel([0.208784, -1.268008, -2.643964, -0.800417, 1.570796, 1.779580],accel_mss,speed_ms,0,blend_radius_m)
    movel([0.208759, -1.266887, -2.644585, -0.800917, 1.570796, 1.779555],accel_mss,speed_ms,0,blend_radius_m)
    movel([0.208572, -1.265804, -2.645183, -0.801402, 1.570796, 1.779369],accel_mss,speed_ms,0,blend_radius_m)
    movel([0.207897, -1.263427, -2.646492, -0.802471, 1.570796, 1.778694],accel_mss,speed_ms,0,blend_radius_m)
    movel([0.207905, -1.262684, -2.646899, -0.802806, 1.570796, 1.778702],accel_mss,speed_ms,0,blend_radius_m)
    movel([0.208101, -1.261942, -2.647305, -0.803142, 1.570796, 1.778897],accel_mss,speed_ms,0,blend_radius_m)
    movel([0.208573, -1.261054, -2.647790, -0.803545, 1.570796, 1.779369],accel_mss,speed_ms,0,blend_radius_m)
    movel([0.209207, -1.260210, -2.648251, -0.803928, 1.570796, 1.780004],accel_mss,speed_ms,0,blend_radius_m)
    movel([0.209973, -1.259432, -2.648675, -0.804283, 1.570796, 1.780769],accel_mss,speed_ms,0,blend_radius_m)
    movel([0.210836, -1.258738, -2.649052, -0.804600, 1.570796, 1.781632],accel_mss,speed_ms,0,blend_radius_m)
    movel([0.211761, -1.258150, -2.649371, -0.804868, 1.570796, 1.782558],accel_mss,speed_ms,0,blend_radius_m)
    movel([0.212715, -1.257690, -2.649620, -0.805079, 1.570796, 1.783511],accel_mss,speed_ms,0,blend_radius_m)
    movel([0.213660, -1.257378, -2.649789, -0.805222, 1.570796, 1.784456],accel_mss,speed_ms,0,blend_radius_m)
    movel([0.214566, -1.257235, -2.649867, -0.805287, 1.570796, 1.785362],accel_mss,speed_ms,0,blend_radius_m)
    movel([0.215386, -1.257282, -2.649841, -0.805266, 1.570796, 1.786182],accel_mss,speed_ms,0,blend_radius_m)
    movel([0.216119, -1.257504, -2.649721, -0.805164, 1.570796, 1.786915],accel_mss,speed_ms,0,blend_radius_m)
    movel([0.216742, -1.257884, -2.649515, -0.804990, 1.570796, 1.787539],accel_mss,speed_ms,0,blend_radius_m)
    movel([0.217226, -1.258400, -2.649235, -0.804754, 1.570796, 1.788023],accel_mss,speed_ms,0,blend_radius_m)
    movel([0.217546, -1.259033, -2.648891, -0.804465, 1.570796, 1.788342],accel_mss,speed_ms,0,blend_radius_m)
    movel([0.217674, -1.259760, -2.648496, -0.804133, 1.570796, 1.788470],accel_mss,speed_ms,0,blend_radius_m)
    movel([0.217589, -1.260561, -2.648059, -0.803768, 1.570796, 1.788386],accel_mss,speed_ms,0,blend_radius_m)
    movel([0.216822, -1.262409, -2.647049, -0.802930, 1.570796, 1.787619],accel_mss,speed_ms,0,blend_radius_m)
    movel([0.216645, -1.263171, -2.646632, -0.802586, 1.570796, 1.787442],accel_mss,speed_ms,0,blend_radius_m)
    movel([0.216707, -1.263743, -2.646318, -0.802328, 1.570796, 1.787504],accel_mss,speed_ms,0,blend_radius_m)
    movel([0.216977, -1.264156, -2.646091, -0.802142, 1.570796, 1.787773],accel_mss,speed_ms,0,blend_radius_m)
    movel([0.218033, -1.264657, -2.645816, -0.801917, 1.570796, 1.788829],accel_mss,speed_ms,0,blend_radius_m)
    movel([0.219586, -1.264961, -2.645648, -0.801780, 1.570796, 1.790383],accel_mss,speed_ms,0,blend_radius_m)
    movel([0.220854, -1.261822, -2.647371, -0.803196, 1.570796, 1.791651],accel_mss,speed_ms,0,blend_radius_m)
    movel([0.221397, -1.260353, -2.648173, -0.803863, 1.570796, 1.792193],accel_mss,speed_ms,0,blend_radius_m)
    movel([0.221758, -1.258952, -2.648935, -0.804501, 1.570796, 1.792554],accel_mss,speed_ms,0,blend_radius_m)
    movel([0.221874, -1.257771, -2.649576, -0.805042, 1.570796, 1.792670],accel_mss,speed_ms,0,blend_radius_m)
    movel([0.221785, -1.256730, -2.650140, -0.805519, 1.570796, 1.792582],accel_mss,speed_ms,0,blend_radius_m)
    movel([0.221506, -1.255822, -2.650630, -0.805937, 1.570796, 1.792302],accel_mss,speed_ms,0,blend_radius_m)
    movel([0.221046, -1.255037, -2.651053, -0.806298, 1.570796, 1.791842],accel_mss,speed_ms,0,blend_radius_m)
    movel([0.220424, -1.254366, -2.651415, -0.806608, 1.570796, 1.791220],accel_mss,speed_ms,0,blend_radius_m)
    movel([0.219648, -1.253804, -2.651717, -0.806868, 1.570796, 1.790445],accel_mss,speed_ms,0,blend_radius_m)
    movel([0.217698, -1.252967, -2.652166, -0.807256, 1.570796, 1.788494],accel_mss,speed_ms,0,blend_radius_m)
    movel([0.222139, -1.248772, -2.654404, -0.809212, 1.570796, 1.792935],accel_mss,speed_ms,0,blend_radius_m)
    movel([0.224204, -1.246619, -2.655545, -0.810225, 1.570796, 1.795001],accel_mss,speed_ms,0,blend_radius_m)
    movel([0.226161, -1.244415, -2.656707, -0.811267, 1.570796, 1.796957],accel_mss,speed_ms,0,blend_radius_m)
    movel([0.228003, -1.242149, -2.657896, -0.812344, 1.570796, 1.798799],accel_mss,speed_ms,0,blend_radius_m)
    movel([0.229726, -1.239812, -2.659115, -0.813461, 1.570796, 1.800523],accel_mss,speed_ms,0,blend_radius_m)
    movel([0.231330, -1.237395, -2.660370, -0.814624, 1.570796, 1.802127],accel_mss,speed_ms,0,blend_radius_m)
    movel([0.232803, -1.234888, -2.661664, -0.815837, 1.570796, 1.803599],accel_mss,speed_ms,0,blend_radius_m)
    movel([0.230920, -1.234418, -2.661906, -0.816065, 1.570796, 1.801717],accel_mss,speed_ms,0,blend_radius_m)
    movel([0.230427, -1.234397, -2.661917, -0.816075, 1.570796, 1.801223],accel_mss,speed_ms,0,blend_radius_m)
    speed_ms = 0.005
    # Splitting Linear movement in 6 (instruction 1375: MoveL 1299)
    movel([0.230427, -1.232785, -2.661145, -0.818459, 1.570796, 1.801223],accel_mss,speed_ms,0,blend_radius_m)
    movel([0.230427, -1.231179, -2.660371, -0.820839, 1.570796, 1.801223],accel_mss,speed_ms,0,blend_radius_m)
    movel([0.230427, -1.229580, -2.659596, -0.823213, 1.570796, 1.801223],accel_mss,speed_ms,0,blend_radius_m)
    movel([0.230427, -1.227987, -2.658819, -0.825583, 1.570796, 1.801223],accel_mss,speed_ms,0,blend_radius_m)
    movel([0.230427, -1.226401, -2.658041, -0.827948, 1.570796, 1.801223],accel_mss,speed_ms,0,blend_radius_m)
    movel([0.230427, -1.224820, -2.657261, -0.830308, 1.570796, 1.801223],accel_mss,speed_ms,0,blend_radius_m)
    speed_ms = 0.040
    # Splitting Linear movement in 6 (instruction 1377: MoveL 1300)
    movel([0.233415, -1.223667, -2.657845, -0.830877, 1.570796, 1.804211],accel_mss,speed_ms,0,blend_radius_m)
    movel([0.236407, -1.222518, -2.658426, -0.831445, 1.570796, 1.807203],accel_mss,speed_ms,0,blend_radius_m)
    movel([0.239402, -1.221373, -2.659003, -0.832013, 1.570796, 1.810198],accel_mss,speed_ms,0,blend_radius_m)
    movel([0.242400, -1.220232, -2.659577, -0.832580, 1.570796, 1.813196],accel_mss,speed_ms,0,blend_radius_m)
    movel([0.245401, -1.219096, -2.660146, -0.833146, 1.570796, 1.816197],accel_mss,speed_ms,0,blend_radius_m)
    movel([0.248406, -1.217965, -2.660712, -0.833712, 1.570796, 1.819202],accel_mss,speed_ms,0,blend_radius_m)
    speed_ms = 0.005
    # Splitting Linear movement in 6 (instruction 1379: MoveL 1301)
    movel([0.248406, -1.219550, -2.661498, -0.831342, 1.570796, 1.819202],accel_mss,speed_ms,0,blend_radius_m)
    movel([0.248406, -1.221141, -2.662281, -0.828967, 1.570796, 1.819202],accel_mss,speed_ms,0,blend_radius_m)
    movel([0.248406, -1.222738, -2.663063, -0.826588, 1.570796, 1.819202],accel_mss,speed_ms,0,blend_radius_m)
    movel([0.248406, -1.224342, -2.663843, -0.824203, 1.570796, 1.819202],accel_mss,speed_ms,0,blend_radius_m)
    movel([0.248406, -1.225953, -2.664622, -0.821814, 1.570796, 1.819202],accel_mss,speed_ms,0,blend_radius_m)
    movel([0.248406, -1.227571, -2.665399, -0.819419, 1.570796, 1.819202],accel_mss,speed_ms,0,blend_radius_m)
    speed_ms = 0.035
    movel([0.249440, -1.227132, -2.665621, -0.819636, 1.570796, 1.820237],accel_mss,speed_ms,0,blend_radius_m)
    movel([0.249896, -1.226652, -2.665864, -0.819873, 1.570796, 1.820692],accel_mss,speed_ms,0,blend_radius_m)
    movel([0.251660, -1.225365, -2.666513, -0.820511, 1.570796, 1.822457],accel_mss,speed_ms,0,blend_radius_m)
    movel([0.252170, -1.224915, -2.666740, -0.820734, 1.570796, 1.822966],accel_mss,speed_ms,0,blend_radius_m)
    movel([0.252526, -1.224419, -2.666989, -0.820981, 1.570796, 1.823322],accel_mss,speed_ms,0,blend_radius_m)
    movel([0.252663, -1.223855, -2.667272, -0.821262, 1.570796, 1.823460],accel_mss,speed_ms,0,blend_radius_m)
    movel([0.252520, -1.223205, -2.667599, -0.821586, 1.570796, 1.823317],accel_mss,speed_ms,0,blend_radius_m)
    movel([0.250957, -1.218948, -2.669722, -0.823719, 1.570796, 1.821754],accel_mss,speed_ms,0,blend_radius_m)
    movel([0.249816, -1.214414, -2.671961, -0.826015, 1.570796, 1.820612],accel_mss,speed_ms,0,blend_radius_m)
    movel([0.249004, -1.209646, -2.674290, -0.828453, 1.570796, 1.819800],accel_mss,speed_ms,0,blend_radius_m)
    movel([0.248438, -1.204690, -2.676684, -0.831015, 1.570796, 1.819234],accel_mss,speed_ms,0,blend_radius_m)
    movel([0.248071, -1.203062, -2.677464, -0.831863, 1.570796, 1.818867],accel_mss,speed_ms,0,blend_radius_m)
    movel([0.247294, -1.201801, -2.678067, -0.832521, 1.570796, 1.818090],accel_mss,speed_ms,0,blend_radius_m)
    movel([0.246094, -1.200947, -2.678474, -0.832968, 1.570796, 1.816891],accel_mss,speed_ms,0,blend_radius_m)
    movel([0.244450, -1.200553, -2.678662, -0.833175, 1.570796, 1.815247],accel_mss,speed_ms,0,blend_radius_m)
    movel([0.243858, -1.200626, -2.678627, -0.833136, 1.570796, 1.814654],accel_mss,speed_ms,0,blend_radius_m)
    movel([0.243176, -1.200861, -2.678515, -0.833013, 1.570796, 1.813973],accel_mss,speed_ms,0,blend_radius_m)
    movel([0.241754, -1.201448, -2.678235, -0.832706, 1.570796, 1.812550],accel_mss,speed_ms,0,blend_radius_m)
    movel([0.241610, -1.203263, -2.677368, -0.831758, 1.570796, 1.812406],accel_mss,speed_ms,0,blend_radius_m)
    movel([0.241596, -1.204126, -2.676954, -0.831308, 1.570796, 1.812393],accel_mss,speed_ms,0,blend_radius_m)
    movel([0.241748, -1.204869, -2.676598, -0.830922, 1.570796, 1.812545],accel_mss,speed_ms,0,blend_radius_m)
    movel([0.242267, -1.205775, -2.676162, -0.830452, 1.570796, 1.813063],accel_mss,speed_ms,0,blend_radius_m)
    movel([0.243552, -1.207402, -2.675377, -0.829610, 1.570796, 1.814349],accel_mss,speed_ms,0,blend_radius_m)
    movel([0.243997, -1.208341, -2.674923, -0.829125, 1.570796, 1.814793],accel_mss,speed_ms,0,blend_radius_m)
    movel([0.244458, -1.211536, -2.673370, -0.827484, 1.570796, 1.815254],accel_mss,speed_ms,0,blend_radius_m)
    movel([0.244873, -1.214752, -2.671794, -0.825843, 1.570796, 1.815669],accel_mss,speed_ms,0,blend_radius_m)
    # Splitting Linear movement in 6 (instruction 1407: MoveL 1328)
    movel([0.245470, -1.216901, -2.670735, -0.824753, 1.570796, 1.816266],accel_mss,speed_ms,0,blend_radius_m)
    movel([0.246063, -1.219044, -2.669674, -0.823671, 1.570796, 1.816859],accel_mss,speed_ms,0,blend_radius_m)
    movel([0.246653, -1.221183, -2.668609, -0.822596, 1.570796, 1.817450],accel_mss,speed_ms,0,blend_radius_m)
    movel([0.247240, -1.223317, -2.667542, -0.821530, 1.570796, 1.818037],accel_mss,speed_ms,0,blend_radius_m)
    movel([0.247825, -1.225446, -2.666472, -0.820470, 1.570796, 1.818621],accel_mss,speed_ms,0,blend_radius_m)
    movel([0.248406, -1.227571, -2.665399, -0.819419, 1.570796, 1.819202],accel_mss,speed_ms,0,blend_radius_m)
    movel([0.249440, -1.227132, -2.665621, -0.819636, 1.570796, 1.820237],accel_mss,speed_ms,0,blend_radius_m)
    movel([0.249896, -1.226652, -2.665864, -0.819873, 1.570796, 1.820692],accel_mss,speed_ms,0,blend_radius_m)
    movel([0.251259, -1.225658, -2.666365, -0.820365, 1.570796, 1.822055],accel_mss,speed_ms,0,blend_radius_m)
    speed_ms = 0.005
    # Splitting Linear movement in 6 (instruction 1412: MoveL 1332)
    movel([0.251259, -1.224040, -2.665587, -0.822763, 1.570796, 1.822055],accel_mss,speed_ms,0,blend_radius_m)
    movel([0.251259, -1.222427, -2.664806, -0.825155, 1.570796, 1.822055],accel_mss,speed_ms,0,blend_radius_m)
    movel([0.251259, -1.220822, -2.664025, -0.827542, 1.570796, 1.822055],accel_mss,speed_ms,0,blend_radius_m)
    movel([0.251259, -1.219223, -2.663241, -0.829925, 1.570796, 1.822055],accel_mss,speed_ms,0,blend_radius_m)
    movel([0.251259, -1.217631, -2.662456, -0.832302, 1.570796, 1.822055],accel_mss,speed_ms,0,blend_radius_m)
    movel([0.251259, -1.216045, -2.661670, -0.834675, 1.570796, 1.822055],accel_mss,speed_ms,0,blend_radius_m)
    speed_ms = 0.040
    # Splitting Linear movement in 14 (instruction 1414: MoveL 1333)
    movel([0.250067, -1.214335, -2.662519, -0.835536, 1.570796, 1.820863],accel_mss,speed_ms,0,blend_radius_m)
    movel([0.248869, -1.212625, -2.663364, -0.836400, 1.570796, 1.819666],accel_mss,speed_ms,0,blend_radius_m)
    movel([0.247667, -1.210914, -2.664207, -0.837268, 1.570796, 1.818463],accel_mss,speed_ms,0,blend_radius_m)
    movel([0.246458, -1.209203, -2.665047, -0.838139, 1.570796, 1.817255],accel_mss,speed_ms,0,blend_radius_m)
    movel([0.245244, -1.207492, -2.665883, -0.839014, 1.570796, 1.816041],accel_mss,speed_ms,0,blend_radius_m)
    movel([0.244025, -1.205780, -2.666716, -0.839892, 1.570796, 1.814821],accel_mss,speed_ms,0,blend_radius_m)
    movel([0.242800, -1.204069, -2.667547, -0.840774, 1.570796, 1.813596],accel_mss,speed_ms,0,blend_radius_m)
    movel([0.241569, -1.202357, -2.668374, -0.841659, 1.570796, 1.812365],accel_mss,speed_ms,0,blend_radius_m)
    movel([0.240332, -1.200645, -2.669198, -0.842547, 1.570796, 1.811129],accel_mss,speed_ms,0,blend_radius_m)
    movel([0.239090, -1.198932, -2.670018, -0.843438, 1.570796, 1.809886],accel_mss,speed_ms,0,blend_radius_m)
    movel([0.237842, -1.197220, -2.670836, -0.844333, 1.570796, 1.808639],accel_mss,speed_ms,0,blend_radius_m)
    movel([0.236589, -1.195508, -2.671650, -0.845231, 1.570796, 1.807385],accel_mss,speed_ms,0,blend_radius_m)
    movel([0.235329, -1.193796, -2.672461, -0.846132, 1.570796, 1.806125],accel_mss,speed_ms,0,blend_radius_m)
    movel([0.234064, -1.192083, -2.673269, -0.847036, 1.570796, 1.804860],accel_mss,speed_ms,0,blend_radius_m)
    speed_ms = 0.005
    # Splitting Linear movement in 6 (instruction 1416: MoveL 1334)
    movel([0.234064, -1.193683, -2.674074, -0.844632, 1.570796, 1.804860],accel_mss,speed_ms,0,blend_radius_m)
    movel([0.234064, -1.195290, -2.674877, -0.842222, 1.570796, 1.804860],accel_mss,speed_ms,0,blend_radius_m)
    movel([0.234064, -1.196904, -2.675678, -0.839807, 1.570796, 1.804860],accel_mss,speed_ms,0,blend_radius_m)
    movel([0.234064, -1.198525, -2.676478, -0.837386, 1.570796, 1.804860],accel_mss,speed_ms,0,blend_radius_m)
    movel([0.234064, -1.200152, -2.677277, -0.834960, 1.570796, 1.804860],accel_mss,speed_ms,0,blend_radius_m)
    movel([0.234064, -1.201787, -2.678074, -0.832528, 1.570796, 1.804860],accel_mss,speed_ms,0,blend_radius_m)
    speed_ms = 0.035
    movel([0.234500, -1.196851, -2.680415, -0.835123, 1.570796, 1.805297],accel_mss,speed_ms,0,blend_radius_m)
    movel([0.234443, -1.195330, -2.681131, -0.835928, 1.570796, 1.805239],accel_mss,speed_ms,0,blend_radius_m)
    movel([0.234120, -1.194957, -2.681307, -0.836126, 1.570796, 1.804916],accel_mss,speed_ms,0,blend_radius_m)
    movel([0.233410, -1.194791, -2.681385, -0.836214, 1.570796, 1.804207],accel_mss,speed_ms,0,blend_radius_m)
    movel([0.231623, -1.194593, -2.681477, -0.836318, 1.570796, 1.802419],accel_mss,speed_ms,0,blend_radius_m)
    movel([0.232111, -1.193134, -2.682161, -0.837094, 1.570796, 1.802907],accel_mss,speed_ms,0,blend_radius_m)
    movel([0.232780, -1.191755, -2.682805, -0.837829, 1.570796, 1.803577],accel_mss,speed_ms,0,blend_radius_m)
    movel([0.233277, -1.191133, -2.683094, -0.838161, 1.570796, 1.804073],accel_mss,speed_ms,0,blend_radius_m)
    movel([0.233931, -1.190581, -2.683351, -0.838457, 1.570796, 1.804728],accel_mss,speed_ms,0,blend_radius_m)
    movel([0.234788, -1.190110, -2.683570, -0.838709, 1.570796, 1.805584],accel_mss,speed_ms,0,blend_radius_m)
    movel([0.236665, -1.189475, -2.683865, -0.839049, 1.570796, 1.807461],accel_mss,speed_ms,0,blend_radius_m)
    movel([0.237415, -1.189101, -2.684038, -0.839250, 1.570796, 1.808212],accel_mss,speed_ms,0,blend_radius_m)
    movel([0.238785, -1.188054, -2.684522, -0.839812, 1.570796, 1.809581],accel_mss,speed_ms,0,blend_radius_m)
    movel([0.239939, -1.186690, -2.685152, -0.840547, 1.570796, 1.810736],accel_mss,speed_ms,0,blend_radius_m)
    movel([0.240846, -1.185083, -2.685891, -0.841415, 1.570796, 1.811642],accel_mss,speed_ms,0,blend_radius_m)
    movel([0.241514, -1.183273, -2.686720, -0.842396, 1.570796, 1.812310],accel_mss,speed_ms,0,blend_radius_m)
    movel([0.241724, -1.181698, -2.687438, -0.843252, 1.570796, 1.812520],accel_mss,speed_ms,0,blend_radius_m)
    movel([0.241632, -1.181010, -2.687751, -0.843628, 1.570796, 1.812428],accel_mss,speed_ms,0,blend_radius_m)
    movel([0.240995, -1.179875, -2.688267, -0.844247, 1.570796, 1.811791],accel_mss,speed_ms,0,blend_radius_m)
    movel([0.240429, -1.179440, -2.688464, -0.844485, 1.570796, 1.811225],accel_mss,speed_ms,0,blend_radius_m)
    movel([0.239616, -1.178840, -2.688736, -0.844814, 1.570796, 1.810413],accel_mss,speed_ms,0,blend_radius_m)
    movel([0.239090, -1.178179, -2.689034, -0.845176, 1.570796, 1.809886],accel_mss,speed_ms,0,blend_radius_m)
    movel([0.238854, -1.177453, -2.689362, -0.845574, 1.570796, 1.809650],accel_mss,speed_ms,0,blend_radius_m)
    movel([0.238909, -1.176649, -2.689724, -0.846016, 1.570796, 1.809705],accel_mss,speed_ms,0,blend_radius_m)
    movel([0.239261, -1.175756, -2.690125, -0.846508, 1.570796, 1.810058],accel_mss,speed_ms,0,blend_radius_m)
    movel([0.239912, -1.174775, -2.690565, -0.847049, 1.570796, 1.810709],accel_mss,speed_ms,0,blend_radius_m)
    movel([0.240863, -1.173690, -2.691051, -0.847648, 1.570796, 1.811659],accel_mss,speed_ms,0,blend_radius_m)
    movel([0.242117, -1.172500, -2.691582, -0.848307, 1.570796, 1.812914],accel_mss,speed_ms,0,blend_radius_m)
    movel([0.243388, -1.171255, -2.692136, -0.848998, 1.570796, 1.814184],accel_mss,speed_ms,0,blend_radius_m)
    movel([0.244363, -1.169984, -2.692700, -0.849705, 1.570796, 1.815160],accel_mss,speed_ms,0,blend_radius_m)
    movel([0.244957, -1.168670, -2.693281, -0.850438, 1.570796, 1.815754],accel_mss,speed_ms,0,blend_radius_m)
    movel([0.245088, -1.167285, -2.693892, -0.851212, 1.570796, 1.815884],accel_mss,speed_ms,0,blend_radius_m)
    movel([0.244714, -1.166203, -2.694367, -0.851819, 1.570796, 1.815511],accel_mss,speed_ms,0,blend_radius_m)
    movel([0.243914, -1.165774, -2.694556, -0.852059, 1.570796, 1.814710],accel_mss,speed_ms,0,blend_radius_m)
    movel([0.242773, -1.165792, -2.694548, -0.852049, 1.570796, 1.813569],accel_mss,speed_ms,0,blend_radius_m)
    movel([0.241377, -1.166055, -2.694433, -0.851902, 1.570796, 1.812174],accel_mss,speed_ms,0,blend_radius_m)
    movel([0.240543, -1.165977, -2.694466, -0.851945, 1.570796, 1.811340],accel_mss,speed_ms,0,blend_radius_m)
    movel([0.239823, -1.165498, -2.694677, -0.852215, 1.570796, 1.810619],accel_mss,speed_ms,0,blend_radius_m)
    movel([0.238377, -1.164191, -2.695249, -0.852949, 1.570796, 1.809174],accel_mss,speed_ms,0,blend_radius_m)
    movel([0.240031, -1.162994, -2.695771, -0.853624, 1.570796, 1.810827],accel_mss,speed_ms,0,blend_radius_m)
    movel([0.241610, -1.162049, -2.696182, -0.854158, 1.570796, 1.812406],accel_mss,speed_ms,0,blend_radius_m)
    movel([0.243098, -1.161351, -2.696485, -0.854552, 1.570796, 1.813894],accel_mss,speed_ms,0,blend_radius_m)
    movel([0.244480, -1.160906, -2.696679, -0.854804, 1.570796, 1.815276],accel_mss,speed_ms,0,blend_radius_m)
    movel([0.245742, -1.160707, -2.696765, -0.854917, 1.570796, 1.816538],accel_mss,speed_ms,0,blend_radius_m)
    movel([0.246865, -1.160755, -2.696744, -0.854890, 1.570796, 1.817661],accel_mss,speed_ms,0,blend_radius_m)
    movel([0.247836, -1.161044, -2.696619, -0.854726, 1.570796, 1.818633],accel_mss,speed_ms,0,blend_radius_m)
    movel([0.248642, -1.161578, -2.696387, -0.854424, 1.570796, 1.819438],accel_mss,speed_ms,0,blend_radius_m)
    movel([0.249310, -1.162397, -2.696031, -0.853961, 1.570796, 1.820106],accel_mss,speed_ms,0,blend_radius_m)
    movel([0.249750, -1.163425, -2.695583, -0.853381, 1.570796, 1.820546],accel_mss,speed_ms,0,blend_radius_m)
    movel([0.249961, -1.164620, -2.695061, -0.852708, 1.570796, 1.820758],accel_mss,speed_ms,0,blend_radius_m)
    movel([0.249947, -1.165930, -2.694487, -0.851972, 1.570796, 1.820743],accel_mss,speed_ms,0,blend_radius_m)
    movel([0.249702, -1.167317, -2.693877, -0.851194, 1.570796, 1.820498],accel_mss,speed_ms,0,blend_radius_m)
    movel([0.249222, -1.168733, -2.693253, -0.850403, 1.570796, 1.820019],accel_mss,speed_ms,0,blend_radius_m)
    movel([0.248507, -1.170140, -2.692631, -0.849618, 1.570796, 1.819303],accel_mss,speed_ms,0,blend_radius_m)
    movel([0.246242, -1.173242, -2.691251, -0.847896, 1.570796, 1.817038],accel_mss,speed_ms,0,blend_radius_m)
    movel([0.245804, -1.174001, -2.690912, -0.847476, 1.570796, 1.816600],accel_mss,speed_ms,0,blend_radius_m)
    movel([0.245520, -1.174703, -2.690598, -0.847089, 1.570796, 1.816316],accel_mss,speed_ms,0,blend_radius_m)
    movel([0.245393, -1.175370, -2.690298, -0.846720, 1.570796, 1.816189],accel_mss,speed_ms,0,blend_radius_m)
    movel([0.245429, -1.176022, -2.690006, -0.846361, 1.570796, 1.816226],accel_mss,speed_ms,0,blend_radius_m)
    movel([0.245998, -1.177353, -2.689407, -0.845629, 1.570796, 1.816794],accel_mss,speed_ms,0,blend_radius_m)
    movel([0.246460, -1.178511, -2.688884, -0.844994, 1.570796, 1.817257],accel_mss,speed_ms,0,blend_radius_m)
    movel([0.246551, -1.179925, -2.688244, -0.844220, 1.570796, 1.817347],accel_mss,speed_ms,0,blend_radius_m)
    movel([0.246303, -1.181531, -2.687514, -0.843343, 1.570796, 1.817100],accel_mss,speed_ms,0,blend_radius_m)
    movel([0.245761, -1.183266, -2.686723, -0.842400, 1.570796, 1.816558],accel_mss,speed_ms,0,blend_radius_m)
    movel([0.244960, -1.185064, -2.685899, -0.841425, 1.570796, 1.815756],accel_mss,speed_ms,0,blend_radius_m)
    movel([0.243935, -1.186869, -2.685070, -0.840451, 1.570796, 1.814732],accel_mss,speed_ms,0,blend_radius_m)
    movel([0.242724, -1.188613, -2.684264, -0.839512, 1.570796, 1.813521],accel_mss,speed_ms,0,blend_radius_m)
    movel([0.241362, -1.190240, -2.683510, -0.838639, 1.570796, 1.812159],accel_mss,speed_ms,0,blend_radius_m)
    movel([0.240644, -1.191131, -2.683096, -0.838163, 1.570796, 1.811440],accel_mss,speed_ms,0,blend_radius_m)
    movel([0.240004, -1.192131, -2.682629, -0.837628, 1.570796, 1.810800],accel_mss,speed_ms,0,blend_radius_m)
    movel([0.239532, -1.193126, -2.682165, -0.837098, 1.570796, 1.810328],accel_mss,speed_ms,0,blend_radius_m)
    movel([0.239311, -1.193994, -2.681758, -0.836636, 1.570796, 1.810108],accel_mss,speed_ms,0,blend_radius_m)
    # Splitting Linear movement in 4 (instruction 1490: MoveL 1407)
    movel([0.239187, -1.195881, -2.680872, -0.835636, 1.570796, 1.809983],accel_mss,speed_ms,0,blend_radius_m)
    movel([0.239063, -1.197762, -2.679985, -0.834642, 1.570796, 1.809859],accel_mss,speed_ms,0,blend_radius_m)
    movel([0.238940, -1.199639, -2.679096, -0.833654, 1.570796, 1.809736],accel_mss,speed_ms,0,blend_radius_m)
    movel([0.238817, -1.201509, -2.678206, -0.832674, 1.570796, 1.809613],accel_mss,speed_ms,0,blend_radius_m)
    # Splitting Linear movement in 4 (instruction 1491: MoveL 1408)
    movel([0.238786, -1.203323, -2.677339, -0.831727, 1.570796, 1.809583],accel_mss,speed_ms,0,blend_radius_m)
    movel([0.238756, -1.205132, -2.676472, -0.830786, 1.570796, 1.809552],accel_mss,speed_ms,0,blend_radius_m)
    movel([0.238726, -1.206936, -2.675602, -0.829851, 1.570796, 1.809522],accel_mss,speed_ms,0,blend_radius_m)
    movel([0.238696, -1.208735, -2.674732, -0.828922, 1.570796, 1.809492],accel_mss,speed_ms,0,blend_radius_m)
    # Splitting Linear movement in 4 (instruction 1492: MoveL 1409)
    movel([0.238761, -1.210476, -2.673886, -0.828027, 1.570796, 1.809558],accel_mss,speed_ms,0,blend_radius_m)
    movel([0.238827, -1.212213, -2.673039, -0.827137, 1.570796, 1.809623],accel_mss,speed_ms,0,blend_radius_m)
    movel([0.238892, -1.213945, -2.672191, -0.826253, 1.570796, 1.809688],accel_mss,speed_ms,0,blend_radius_m)
    movel([0.238956, -1.215673, -2.671341, -0.825375, 1.570796, 1.809753],accel_mss,speed_ms,0,blend_radius_m)
    # Splitting Linear movement in 4 (instruction 1493: MoveL 1410)
    movel([0.239121, -1.217341, -2.670518, -0.824530, 1.570796, 1.809917],accel_mss,speed_ms,0,blend_radius_m)
    movel([0.239285, -1.219005, -2.669693, -0.823690, 1.570796, 1.810082],accel_mss,speed_ms,0,blend_radius_m)
    movel([0.239449, -1.220666, -2.668867, -0.822856, 1.570796, 1.810245],accel_mss,speed_ms,0,blend_radius_m)
    movel([0.239612, -1.222323, -2.668040, -0.822026, 1.570796, 1.810408],accel_mss,speed_ms,0,blend_radius_m)
    # Splitting Linear movement in 4 (instruction 1494: MoveL 1411)
    movel([0.239879, -1.223919, -2.667240, -0.821230, 1.570796, 1.810675],accel_mss,speed_ms,0,blend_radius_m)
    movel([0.240145, -1.225512, -2.666439, -0.820438, 1.570796, 1.810941],accel_mss,speed_ms,0,blend_radius_m)
    movel([0.240410, -1.227102, -2.665637, -0.819651, 1.570796, 1.811206],accel_mss,speed_ms,0,blend_radius_m)
    movel([0.240674, -1.228688, -2.664833, -0.818868, 1.570796, 1.811470],accel_mss,speed_ms,0,blend_radius_m)
    # Splitting Linear movement in 4 (instruction 1495: MoveL 1412)
    movel([0.241047, -1.230211, -2.664059, -0.818119, 1.570796, 1.811844],accel_mss,speed_ms,0,blend_radius_m)
    movel([0.241419, -1.231730, -2.663284, -0.817375, 1.570796, 1.812216],accel_mss,speed_ms,0,blend_radius_m)
    movel([0.241790, -1.233247, -2.662507, -0.816634, 1.570796, 1.812586],accel_mss,speed_ms,0,blend_radius_m)
    movel([0.242159, -1.234762, -2.661729, -0.815898, 1.570796, 1.812955],accel_mss,speed_ms,0,blend_radius_m)
    # Splitting Linear movement in 4 (instruction 1496: MoveL 1413)
    movel([0.242641, -1.236212, -2.660982, -0.815195, 1.570796, 1.813438],accel_mss,speed_ms,0,blend_radius_m)
    movel([0.243122, -1.237660, -2.660233, -0.814496, 1.570796, 1.813918],accel_mss,speed_ms,0,blend_radius_m)
    movel([0.243601, -1.239106, -2.659483, -0.813800, 1.570796, 1.814397],accel_mss,speed_ms,0,blend_radius_m)
    movel([0.244078, -1.240550, -2.658731, -0.813108, 1.570796, 1.814874],accel_mss,speed_ms,0,blend_radius_m)
    # Splitting Linear movement in 4 (instruction 1497: MoveL 1414)
    movel([0.244672, -1.241928, -2.658012, -0.812450, 1.570796, 1.815469],accel_mss,speed_ms,0,blend_radius_m)
    movel([0.245265, -1.243304, -2.657291, -0.811794, 1.570796, 1.816061],accel_mss,speed_ms,0,blend_radius_m)
    movel([0.245855, -1.244678, -2.656569, -0.811142, 1.570796, 1.816651],accel_mss,speed_ms,0,blend_radius_m)
    movel([0.246443, -1.246052, -2.655845, -0.810492, 1.570796, 1.817239],accel_mss,speed_ms,0,blend_radius_m)
    movel([0.247763, -1.248596, -2.654498, -0.809295, 1.570796, 1.818559],accel_mss,speed_ms,0,blend_radius_m)
    movel([0.244037, -1.251821, -2.652780, -0.807789, 1.570796, 1.814834],accel_mss,speed_ms,0,blend_radius_m)
    movel([0.242518, -1.249506, -2.654014, -0.808869, 1.570796, 1.813314],accel_mss,speed_ms,0,blend_radius_m)
    # Splitting Linear movement in 4 (instruction 1501: MoveL 1418)
    movel([0.242021, -1.248410, -2.654597, -0.809382, 1.570796, 1.812817],accel_mss,speed_ms,0,blend_radius_m)
    movel([0.241523, -1.247313, -2.655178, -0.809898, 1.570796, 1.812319],accel_mss,speed_ms,0,blend_radius_m)
    movel([0.241023, -1.246215, -2.655759, -0.810415, 1.570796, 1.811819],accel_mss,speed_ms,0,blend_radius_m)
    movel([0.240522, -1.245116, -2.656338, -0.810935, 1.570796, 1.811318],accel_mss,speed_ms,0,blend_radius_m)
    # Splitting Linear movement in 4 (instruction 1502: MoveL 1419)
    movel([0.240094, -1.243973, -2.656940, -0.811477, 1.570796, 1.810890],accel_mss,speed_ms,0,blend_radius_m)
    movel([0.239664, -1.242828, -2.657541, -0.812021, 1.570796, 1.810460],accel_mss,speed_ms,0,blend_radius_m)
    movel([0.239233, -1.241682, -2.658140, -0.812567, 1.570796, 1.810030],accel_mss,speed_ms,0,blend_radius_m)
    movel([0.238801, -1.240534, -2.658739, -0.813115, 1.570796, 1.809597],accel_mss,speed_ms,0,blend_radius_m)
    # Splitting Linear movement in 4 (instruction 1503: MoveL 1420)
    movel([0.238439, -1.239345, -2.659359, -0.813686, 1.570796, 1.809236],accel_mss,speed_ms,0,blend_radius_m)
    movel([0.238077, -1.238153, -2.659977, -0.814258, 1.570796, 1.808873],accel_mss,speed_ms,0,blend_radius_m)
    movel([0.237713, -1.236961, -2.660595, -0.814833, 1.570796, 1.808509],accel_mss,speed_ms,0,blend_radius_m)
    movel([0.237348, -1.235766, -2.661212, -0.815411, 1.570796, 1.808144],accel_mss,speed_ms,0,blend_radius_m)
    # Splitting Linear movement in 4 (instruction 1504: MoveL 1421)
    movel([0.237052, -1.234528, -2.661849, -0.816012, 1.570796, 1.807848],accel_mss,speed_ms,0,blend_radius_m)
    movel([0.236755, -1.233288, -2.662486, -0.816615, 1.570796, 1.807551],accel_mss,speed_ms,0,blend_radius_m)
    movel([0.236457, -1.232046, -2.663122, -0.817221, 1.570796, 1.807254],accel_mss,speed_ms,0,blend_radius_m)
    movel([0.236159, -1.230803, -2.663757, -0.817829, 1.570796, 1.806955],accel_mss,speed_ms,0,blend_radius_m)
    # Splitting Linear movement in 4 (instruction 1505: MoveL 1422)
    movel([0.235926, -1.229517, -2.664412, -0.818460, 1.570796, 1.806723],accel_mss,speed_ms,0,blend_radius_m)
    movel([0.235693, -1.228230, -2.665065, -0.819093, 1.570796, 1.806489],accel_mss,speed_ms,0,blend_radius_m)
    movel([0.235459, -1.226941, -2.665718, -0.819730, 1.570796, 1.806255],accel_mss,speed_ms,0,blend_radius_m)
    movel([0.235224, -1.225650, -2.666369, -0.820369, 1.570796, 1.806021],accel_mss,speed_ms,0,blend_radius_m)
    # Splitting Linear movement in 4 (instruction 1506: MoveL 1423)
    movel([0.235055, -1.224318, -2.667040, -0.821031, 1.570796, 1.805852],accel_mss,speed_ms,0,blend_radius_m)
    movel([0.234886, -1.222983, -2.667710, -0.821696, 1.570796, 1.805682],accel_mss,speed_ms,0,blend_radius_m)
    movel([0.234716, -1.221646, -2.668379, -0.822365, 1.570796, 1.805512],accel_mss,speed_ms,0,blend_radius_m)
    movel([0.234545, -1.220306, -2.669046, -0.823036, 1.570796, 1.805341],accel_mss,speed_ms,0,blend_radius_m)
    # Splitting Linear movement in 4 (instruction 1507: MoveL 1424)
    movel([0.234437, -1.218925, -2.669733, -0.823731, 1.570796, 1.805233],accel_mss,speed_ms,0,blend_radius_m)
    movel([0.234328, -1.217542, -2.670418, -0.824429, 1.570796, 1.805125],accel_mss,speed_ms,0,blend_radius_m)
    movel([0.234220, -1.216156, -2.671103, -0.825130, 1.570796, 1.805016],accel_mss,speed_ms,0,blend_radius_m)
    movel([0.234110, -1.214768, -2.671786, -0.825835, 1.570796, 1.804907],accel_mss,speed_ms,0,blend_radius_m)
    # Splitting Linear movement in 4 (instruction 1508: MoveL 1425)
    movel([0.234063, -1.212890, -2.672707, -0.826791, 1.570796, 1.804859],accel_mss,speed_ms,0,blend_radius_m)
    movel([0.234015, -1.211008, -2.673627, -0.827754, 1.570796, 1.804812],accel_mss,speed_ms,0,blend_radius_m)
    movel([0.233968, -1.209120, -2.674545, -0.828724, 1.570796, 1.804764],accel_mss,speed_ms,0,blend_radius_m)
    movel([0.233920, -1.207228, -2.675461, -0.829700, 1.570796, 1.804716],accel_mss,speed_ms,0,blend_radius_m)
    movel([0.233769, -1.206898, -2.675621, -0.829870, 1.570796, 1.804565],accel_mss,speed_ms,0,blend_radius_m)
    movel([0.233476, -1.206688, -2.675722, -0.829979, 1.570796, 1.804273],accel_mss,speed_ms,0,blend_radius_m)
    movel([0.233010, -1.206622, -2.675754, -0.830013, 1.570796, 1.803807],accel_mss,speed_ms,0,blend_radius_m)
    movel([0.232321, -1.206744, -2.675695, -0.829950, 1.570796, 1.803117],accel_mss,speed_ms,0,blend_radius_m)
    movel([0.231007, -1.207260, -2.675446, -0.829683, 1.570796, 1.801803],accel_mss,speed_ms,0,blend_radius_m)
    movel([0.229895, -1.208028, -2.675074, -0.829287, 1.570796, 1.800692],accel_mss,speed_ms,0,blend_radius_m)
    movel([0.228998, -1.209036, -2.674586, -0.828767, 1.570796, 1.799794],accel_mss,speed_ms,0,blend_radius_m)
    movel([0.228318, -1.210282, -2.673981, -0.828127, 1.570796, 1.799114],accel_mss,speed_ms,0,blend_radius_m)
    movel([0.227837, -1.211601, -2.673338, -0.827450, 1.570796, 1.798634],accel_mss,speed_ms,0,blend_radius_m)
    movel([0.227647, -1.212779, -2.672762, -0.826848, 1.570796, 1.798443],accel_mss,speed_ms,0,blend_radius_m)
    movel([0.227907, -1.213723, -2.672300, -0.826367, 1.570796, 1.798703],accel_mss,speed_ms,0,blend_radius_m)
    movel([0.228774, -1.214349, -2.671992, -0.826048, 1.570796, 1.799570],accel_mss,speed_ms,0,blend_radius_m)
    movel([0.229795, -1.214794, -2.671774, -0.825821, 1.570796, 1.800591],accel_mss,speed_ms,0,blend_radius_m)
    movel([0.230184, -1.215118, -2.671614, -0.825657, 1.570796, 1.800980],accel_mss,speed_ms,0,blend_radius_m)
    movel([0.230360, -1.215549, -2.671402, -0.825438, 1.570796, 1.801156],accel_mss,speed_ms,0,blend_radius_m)
    movel([0.230272, -1.216981, -2.670696, -0.824712, 1.570796, 1.801068],accel_mss,speed_ms,0,blend_radius_m)
    movel([0.230056, -1.217528, -2.670425, -0.824436, 1.570796, 1.800852],accel_mss,speed_ms,0,blend_radius_m)
    movel([0.229722, -1.217966, -2.670208, -0.824214, 1.570796, 1.800518],accel_mss,speed_ms,0,blend_radius_m)
    movel([0.229267, -1.218306, -2.670040, -0.824043, 1.570796, 1.800063],accel_mss,speed_ms,0,blend_radius_m)
    movel([0.228687, -1.218550, -2.669919, -0.823920, 1.570796, 1.799483],accel_mss,speed_ms,0,blend_radius_m)
    movel([0.227147, -1.218772, -2.669809, -0.823808, 1.570796, 1.797944],accel_mss,speed_ms,0,blend_radius_m)
    movel([0.226102, -1.218711, -2.669839, -0.823839, 1.570796, 1.796899],accel_mss,speed_ms,0,blend_radius_m)
    movel([0.225205, -1.218469, -2.669959, -0.823961, 1.570796, 1.796002],accel_mss,speed_ms,0,blend_radius_m)
    movel([0.224464, -1.218051, -2.670166, -0.824171, 1.570796, 1.795260],accel_mss,speed_ms,0,blend_radius_m)
    movel([0.223884, -1.217462, -2.670458, -0.824469, 1.570796, 1.794681],accel_mss,speed_ms,0,blend_radius_m)
    movel([0.223471, -1.216709, -2.670830, -0.824850, 1.570796, 1.794268],accel_mss,speed_ms,0,blend_radius_m)
    movel([0.223231, -1.215799, -2.671279, -0.825311, 1.570796, 1.794028],accel_mss,speed_ms,0,blend_radius_m)
    movel([0.223169, -1.214737, -2.671802, -0.825850, 1.570796, 1.793965],accel_mss,speed_ms,0,blend_radius_m)
    movel([0.223291, -1.213532, -2.672393, -0.826464, 1.570796, 1.794087],accel_mss,speed_ms,0,blend_radius_m)
    movel([0.223636, -1.212033, -2.673127, -0.827229, 1.570796, 1.794432],accel_mss,speed_ms,0,blend_radius_m)
    movel([0.224145, -1.210584, -2.673834, -0.827972, 1.570796, 1.794941],accel_mss,speed_ms,0,blend_radius_m)
    movel([0.224811, -1.209198, -2.674507, -0.828684, 1.570796, 1.795607],accel_mss,speed_ms,0,blend_radius_m)
    movel([0.225622, -1.207895, -2.675139, -0.829355, 1.570796, 1.796419],accel_mss,speed_ms,0,blend_radius_m)
    movel([0.226575, -1.206681, -2.675725, -0.829983, 1.570796, 1.797371],accel_mss,speed_ms,0,blend_radius_m)
    movel([0.227656, -1.205577, -2.676257, -0.830555, 1.570796, 1.798452],accel_mss,speed_ms,0,blend_radius_m)
    movel([0.228860, -1.204591, -2.676731, -0.831067, 1.570796, 1.799657],accel_mss,speed_ms,0,blend_radius_m)
    movel([0.230174, -1.203747, -2.677136, -0.831506, 1.570796, 1.800970],accel_mss,speed_ms,0,blend_radius_m)
    movel([0.234064, -1.201787, -2.678074, -0.832528, 1.570796, 1.804860],accel_mss,speed_ms,0,blend_radius_m)
    movel([0.234315, -1.198969, -2.679414, -0.834006, 1.570796, 1.805111],accel_mss,speed_ms,0,blend_radius_m)
    speed_ms = 0.005
    # Splitting Linear movement in 4 (instruction 1549: MoveL 1465)
    movel([0.234315, -1.196517, -2.678215, -0.837657, 1.570796, 1.805111],accel_mss,speed_ms,0,blend_radius_m)
    movel([0.234315, -1.194081, -2.677012, -0.841296, 1.570796, 1.805111],accel_mss,speed_ms,0,blend_radius_m)
    movel([0.234315, -1.191661, -2.675806, -0.844922, 1.570796, 1.805111],accel_mss,speed_ms,0,blend_radius_m)
    movel([0.234315, -1.189256, -2.674597, -0.848536, 1.570796, 1.805111],accel_mss,speed_ms,0,blend_radius_m)
    speed_ms = 0.040
    # Splitting Linear movement in 14 (instruction 1551: MoveL 1466)
    movel([0.232982, -1.187792, -2.675281, -0.849317, 1.570796, 1.803778],accel_mss,speed_ms,0,blend_radius_m)
    movel([0.231644, -1.186328, -2.675962, -0.850099, 1.570796, 1.802440],accel_mss,speed_ms,0,blend_radius_m)
    movel([0.230300, -1.184866, -2.676640, -0.850883, 1.570796, 1.801096],accel_mss,speed_ms,0,blend_radius_m)
    movel([0.228950, -1.183405, -2.677316, -0.851668, 1.570796, 1.799747],accel_mss,speed_ms,0,blend_radius_m)
    movel([0.227595, -1.181946, -2.677988, -0.852455, 1.570796, 1.798392],accel_mss,speed_ms,0,blend_radius_m)
    movel([0.226235, -1.180488, -2.678658, -0.853243, 1.570796, 1.797031],accel_mss,speed_ms,0,blend_radius_m)
    movel([0.224869, -1.179031, -2.679325, -0.854033, 1.570796, 1.795665],accel_mss,speed_ms,0,blend_radius_m)
    movel([0.223497, -1.177575, -2.679989, -0.854825, 1.570796, 1.794293],accel_mss,speed_ms,0,blend_radius_m)
    movel([0.222120, -1.176121, -2.680650, -0.855618, 1.570796, 1.792916],accel_mss,speed_ms,0,blend_radius_m)
    movel([0.220737, -1.174668, -2.681308, -0.856412, 1.570796, 1.791533],accel_mss,speed_ms,0,blend_radius_m)
    movel([0.219348, -1.173217, -2.681964, -0.857208, 1.570796, 1.790144],accel_mss,speed_ms,0,blend_radius_m)
    movel([0.217954, -1.171767, -2.682616, -0.858005, 1.570796, 1.788750],accel_mss,speed_ms,0,blend_radius_m)
    movel([0.216554, -1.170319, -2.683266, -0.858804, 1.570796, 1.787350],accel_mss,speed_ms,0,blend_radius_m)
    movel([0.215148, -1.168873, -2.683913, -0.859603, 1.570796, 1.785944],accel_mss,speed_ms,0,blend_radius_m)
    speed_ms = 0.005
    # Splitting Linear movement in 6 (instruction 1553: MoveL 1467)
    movel([0.215148, -1.170484, -2.684735, -0.857170, 1.570796, 1.785944],accel_mss,speed_ms,0,blend_radius_m)
    movel([0.215148, -1.172103, -2.685555, -0.854731, 1.570796, 1.785944],accel_mss,speed_ms,0,blend_radius_m)
    movel([0.215148, -1.173728, -2.686374, -0.852287, 1.570796, 1.785944],accel_mss,speed_ms,0,blend_radius_m)
    movel([0.215148, -1.175361, -2.687191, -0.849836, 1.570796, 1.785944],accel_mss,speed_ms,0,blend_radius_m)
    movel([0.215148, -1.177002, -2.688007, -0.847380, 1.570796, 1.785944],accel_mss,speed_ms,0,blend_radius_m)
    movel([0.215148, -1.178649, -2.688822, -0.844918, 1.570796, 1.785944],accel_mss,speed_ms,0,blend_radius_m)
    speed_ms = 0.035
    movel([0.215496, -1.179911, -2.688250, -0.844228, 1.570796, 1.786292],accel_mss,speed_ms,0,blend_radius_m)
    movel([0.215567, -1.181152, -2.687687, -0.843550, 1.570796, 1.786364],accel_mss,speed_ms,0,blend_radius_m)
    movel([0.215364, -1.181815, -2.687385, -0.843189, 1.570796, 1.786160],accel_mss,speed_ms,0,blend_radius_m)
    movel([0.214937, -1.182529, -2.687060, -0.842801, 1.570796, 1.785734],accel_mss,speed_ms,0,blend_radius_m)
    movel([0.214225, -1.183314, -2.686701, -0.842374, 1.570796, 1.785022],accel_mss,speed_ms,0,blend_radius_m)
    movel([0.213184, -1.184189, -2.686301, -0.841899, 1.570796, 1.783980],accel_mss,speed_ms,0,blend_radius_m)
    movel([0.212418, -1.184898, -2.685976, -0.841515, 1.570796, 1.783214],accel_mss,speed_ms,0,blend_radius_m)
    movel([0.211892, -1.185666, -2.685623, -0.841100, 1.570796, 1.782688],accel_mss,speed_ms,0,blend_radius_m)
    movel([0.211594, -1.186454, -2.685261, -0.840674, 1.570796, 1.782390],accel_mss,speed_ms,0,blend_radius_m)
    movel([0.211512, -1.187231, -2.684902, -0.840255, 1.570796, 1.782308],accel_mss,speed_ms,0,blend_radius_m)
    movel([0.211641, -1.187960, -2.684566, -0.839863, 1.570796, 1.782437],accel_mss,speed_ms,0,blend_radius_m)
    movel([0.211965, -1.188612, -2.684265, -0.839513, 1.570796, 1.782761],accel_mss,speed_ms,0,blend_radius_m)
    movel([0.212481, -1.189151, -2.684015, -0.839223, 1.570796, 1.783277],accel_mss,speed_ms,0,blend_radius_m)
    movel([0.213179, -1.189544, -2.683833, -0.839012, 1.570796, 1.783975],accel_mss,speed_ms,0,blend_radius_m)
    movel([0.216880, -1.191013, -2.683150, -0.838225, 1.570796, 1.787677],accel_mss,speed_ms,0,blend_radius_m)
    movel([0.218608, -1.191888, -2.682743, -0.837758, 1.570796, 1.789405],accel_mss,speed_ms,0,blend_radius_m)
    movel([0.220133, -1.192972, -2.682237, -0.837180, 1.570796, 1.790929],accel_mss,speed_ms,0,blend_radius_m)
    movel([0.221025, -1.193870, -2.681817, -0.836703, 1.570796, 1.791821],accel_mss,speed_ms,0,blend_radius_m)
    movel([0.222367, -1.195964, -2.680833, -0.835592, 1.570796, 1.793164],accel_mss,speed_ms,0,blend_radius_m)
    movel([0.222822, -1.197146, -2.680276, -0.834967, 1.570796, 1.793618],accel_mss,speed_ms,0,blend_radius_m)
    movel([0.223312, -1.199735, -2.679050, -0.833604, 1.570796, 1.794108],accel_mss,speed_ms,0,blend_radius_m)
    movel([0.223348, -1.201129, -2.678387, -0.832873, 1.570796, 1.794145],accel_mss,speed_ms,0,blend_radius_m)
    movel([0.223248, -1.202582, -2.677694, -0.832113, 1.570796, 1.794045],accel_mss,speed_ms,0,blend_radius_m)
    movel([0.222651, -1.205623, -2.676235, -0.830531, 1.570796, 1.793447],accel_mss,speed_ms,0,blend_radius_m)
    movel([0.221536, -1.208807, -2.674697, -0.828885, 1.570796, 1.792332],accel_mss,speed_ms,0,blend_radius_m)
    movel([0.219921, -1.212072, -2.673108, -0.827209, 1.570796, 1.790717],accel_mss,speed_ms,0,blend_radius_m)
    movel([0.217815, -1.215368, -2.671491, -0.825530, 1.570796, 1.788612],accel_mss,speed_ms,0,blend_radius_m)
    movel([0.217091, -1.216477, -2.670945, -0.824967, 1.570796, 1.787887],accel_mss,speed_ms,0,blend_radius_m)
    movel([0.216507, -1.217552, -2.670414, -0.824424, 1.570796, 1.787303],accel_mss,speed_ms,0,blend_radius_m)
    movel([0.215752, -1.219566, -2.669415, -0.823408, 1.570796, 1.786548],accel_mss,speed_ms,0,blend_radius_m)
    movel([0.215530, -1.221354, -2.668524, -0.822511, 1.570796, 1.786326],accel_mss,speed_ms,0,blend_radius_m)
    movel([0.215812, -1.222860, -2.667771, -0.821758, 1.570796, 1.786608],accel_mss,speed_ms,0,blend_radius_m)
    movel([0.216570, -1.224025, -2.667187, -0.821177, 1.570796, 1.787367],accel_mss,speed_ms,0,blend_radius_m)
    movel([0.217786, -1.224795, -2.666800, -0.820794, 1.570796, 1.788583],accel_mss,speed_ms,0,blend_radius_m)
    movel([0.219430, -1.225111, -2.666641, -0.820637, 1.570796, 1.790226],accel_mss,speed_ms,0,blend_radius_m)
    movel([0.220408, -1.225080, -2.666657, -0.820653, 1.570796, 1.791205],accel_mss,speed_ms,0,blend_radius_m)
    movel([0.222956, -1.224582, -2.666907, -0.820900, 1.570796, 1.793752],accel_mss,speed_ms,0,blend_radius_m)
    movel([0.224445, -1.224089, -2.667155, -0.821145, 1.570796, 1.795242],accel_mss,speed_ms,0,blend_radius_m)
    movel([0.225247, -1.223820, -2.667290, -0.821279, 1.570796, 1.796043],accel_mss,speed_ms,0,blend_radius_m)
    movel([0.225834, -1.223757, -2.667321, -0.821310, 1.570796, 1.796630],accel_mss,speed_ms,0,blend_radius_m)
    movel([0.226243, -1.223870, -2.667265, -0.821254, 1.570796, 1.797039],accel_mss,speed_ms,0,blend_radius_m)
    movel([0.226496, -1.224132, -2.667133, -0.821124, 1.570796, 1.797293],accel_mss,speed_ms,0,blend_radius_m)
    movel([0.226664, -1.224974, -2.666710, -0.820705, 1.570796, 1.797461],accel_mss,speed_ms,0,blend_radius_m)
    movel([0.226566, -1.226049, -2.666168, -0.820172, 1.570796, 1.797362],accel_mss,speed_ms,0,blend_radius_m)
    movel([0.226415, -1.226636, -2.665872, -0.819881, 1.570796, 1.797211],accel_mss,speed_ms,0,blend_radius_m)
    movel([0.226168, -1.227092, -2.665642, -0.819655, 1.570796, 1.796964],accel_mss,speed_ms,0,blend_radius_m)
    movel([0.225458, -1.227695, -2.665336, -0.819357, 1.570796, 1.796254],accel_mss,speed_ms,0,blend_radius_m)
    movel([0.224613, -1.228005, -2.665180, -0.819205, 1.570796, 1.795410],accel_mss,speed_ms,0,blend_radius_m)
    movel([0.219938, -1.229000, -2.664675, -0.818715, 1.570796, 1.790735],accel_mss,speed_ms,0,blend_radius_m)
    movel([0.218064, -1.229272, -2.664536, -0.818580, 1.570796, 1.788861],accel_mss,speed_ms,0,blend_radius_m)
    movel([0.216326, -1.229305, -2.664520, -0.818564, 1.570796, 1.787122],accel_mss,speed_ms,0,blend_radius_m)
    movel([0.215237, -1.229140, -2.664604, -0.818646, 1.570796, 1.786034],accel_mss,speed_ms,0,blend_radius_m)
    movel([0.214274, -1.228820, -2.664766, -0.818803, 1.570796, 1.785071],accel_mss,speed_ms,0,blend_radius_m)
    movel([0.213435, -1.228357, -2.665001, -0.819031, 1.570796, 1.784231],accel_mss,speed_ms,0,blend_radius_m)
    movel([0.212132, -1.227049, -2.665663, -0.819677, 1.570796, 1.782928],accel_mss,speed_ms,0,blend_radius_m)
    movel([0.211669, -1.226224, -2.666080, -0.820085, 1.570796, 1.782466],accel_mss,speed_ms,0,blend_radius_m)
    movel([0.211129, -1.224298, -2.667050, -0.821041, 1.570796, 1.781926],accel_mss,speed_ms,0,blend_radius_m)
    movel([0.211054, -1.223213, -2.667594, -0.821582, 1.570796, 1.781850],accel_mss,speed_ms,0,blend_radius_m)
    movel([0.211301, -1.220865, -2.668768, -0.822756, 1.570796, 1.782097],accel_mss,speed_ms,0,blend_radius_m)
    movel([0.211629, -1.219619, -2.669388, -0.823381, 1.570796, 1.782426],accel_mss,speed_ms,0,blend_radius_m)
    movel([0.212696, -1.217054, -2.670660, -0.824675, 1.570796, 1.783492],accel_mss,speed_ms,0,blend_radius_m)
    movel([0.213436, -1.215756, -2.671300, -0.825333, 1.570796, 1.784233],accel_mss,speed_ms,0,blend_radius_m)
    movel([0.215990, -1.211955, -2.673165, -0.827269, 1.570796, 1.786786],accel_mss,speed_ms,0,blend_radius_m)
    movel([0.217288, -1.209456, -2.674382, -0.828551, 1.570796, 1.788085],accel_mss,speed_ms,0,blend_radius_m)
    movel([0.218199, -1.207015, -2.675564, -0.829810, 1.570796, 1.788995],accel_mss,speed_ms,0,blend_radius_m)
    movel([0.218709, -1.204671, -2.676693, -0.831025, 1.570796, 1.789506],accel_mss,speed_ms,0,blend_radius_m)
    movel([0.218807, -1.202470, -2.677747, -0.832172, 1.570796, 1.789603],accel_mss,speed_ms,0,blend_radius_m)
    movel([0.218474, -1.200465, -2.678704, -0.833221, 1.570796, 1.789270],accel_mss,speed_ms,0,blend_radius_m)
    movel([0.217699, -1.198697, -2.679543, -0.834149, 1.570796, 1.788495],accel_mss,speed_ms,0,blend_radius_m)
    movel([0.216465, -1.197220, -2.680241, -0.834928, 1.570796, 1.787262],accel_mss,speed_ms,0,blend_radius_m)
    movel([0.215129, -1.196214, -2.680715, -0.835459, 1.570796, 1.785926],accel_mss,speed_ms,0,blend_radius_m)
    movel([0.213608, -1.195393, -2.681102, -0.835894, 1.570796, 1.784405],accel_mss,speed_ms,0,blend_radius_m)
    movel([0.209305, -1.193766, -2.681865, -0.836758, 1.570796, 1.780101],accel_mss,speed_ms,0,blend_radius_m)
    movel([0.208498, -1.193233, -2.682115, -0.837041, 1.570796, 1.779294],accel_mss,speed_ms,0,blend_radius_m)
    movel([0.207839, -1.192553, -2.682432, -0.837403, 1.570796, 1.778636],accel_mss,speed_ms,0,blend_radius_m)
    movel([0.207340, -1.191735, -2.682814, -0.837840, 1.570796, 1.778136],accel_mss,speed_ms,0,blend_radius_m)
    movel([0.207014, -1.190786, -2.683256, -0.838347, 1.570796, 1.777811],accel_mss,speed_ms,0,blend_radius_m)
    movel([0.206876, -1.189713, -2.683755, -0.838922, 1.570796, 1.777673],accel_mss,speed_ms,0,blend_radius_m)
    movel([0.206937, -1.188523, -2.684306, -0.839560, 1.570796, 1.777733],accel_mss,speed_ms,0,blend_radius_m)
    movel([0.207215, -1.187222, -2.684907, -0.840260, 1.570796, 1.778011],accel_mss,speed_ms,0,blend_radius_m)
    movel([0.207644, -1.186014, -2.685463, -0.840912, 1.570796, 1.778441],accel_mss,speed_ms,0,blend_radius_m)
    movel([0.208236, -1.184838, -2.686003, -0.841547, 1.570796, 1.779032],accel_mss,speed_ms,0,blend_radius_m)
    movel([0.208985, -1.183701, -2.686524, -0.842164, 1.570796, 1.779782],accel_mss,speed_ms,0,blend_radius_m)
    movel([0.209896, -1.182602, -2.687026, -0.842760, 1.570796, 1.780693],accel_mss,speed_ms,0,blend_radius_m)
    movel([0.210965, -1.181546, -2.687507, -0.843335, 1.570796, 1.781762],accel_mss,speed_ms,0,blend_radius_m)
    movel([0.212199, -1.180531, -2.687969, -0.843889, 1.570796, 1.782995],accel_mss,speed_ms,0,blend_radius_m)
    movel([0.213592, -1.179566, -2.688407, -0.844416, 1.570796, 1.784388],accel_mss,speed_ms,0,blend_radius_m)
    movel([0.215148, -1.178649, -2.688822, -0.844918, 1.570796, 1.785944],accel_mss,speed_ms,0,blend_radius_m)
    movel([0.215496, -1.179911, -2.688250, -0.844228, 1.570796, 1.786292],accel_mss,speed_ms,0,blend_radius_m)
    movel([0.215567, -1.181152, -2.687687, -0.843550, 1.570796, 1.786364],accel_mss,speed_ms,0,blend_radius_m)
    speed_ms = 0.005
    # Splitting Linear movement in 6 (instruction 1646: MoveL 1558)
    movel([0.215567, -1.179506, -2.686874, -0.846009, 1.570796, 1.786364],accel_mss,speed_ms,0,blend_radius_m)
    movel([0.215567, -1.177867, -2.686060, -0.848462, 1.570796, 1.786364],accel_mss,speed_ms,0,blend_radius_m)
    movel([0.215567, -1.176235, -2.685245, -0.850909, 1.570796, 1.786364],accel_mss,speed_ms,0,blend_radius_m)
    movel([0.215567, -1.174611, -2.684428, -0.853351, 1.570796, 1.786364],accel_mss,speed_ms,0,blend_radius_m)
    movel([0.215567, -1.172993, -2.683609, -0.855787, 1.570796, 1.786364],accel_mss,speed_ms,0,blend_radius_m)
    movel([0.215567, -1.171383, -2.682789, -0.858217, 1.570796, 1.786364],accel_mss,speed_ms,0,blend_radius_m)
    speed_ms = 0.040
    # Splitting Linear movement in 12 (instruction 1648: MoveL 1559)
    movel([0.217405, -1.168320, -2.684160, -0.859910, 1.570796, 1.788201],accel_mss,speed_ms,0,blend_radius_m)
    movel([0.219253, -1.165241, -2.685527, -0.861621, 1.570796, 1.790049],accel_mss,speed_ms,0,blend_radius_m)
    movel([0.221112, -1.162146, -2.686892, -0.863351, 1.570796, 1.791908],accel_mss,speed_ms,0,blend_radius_m)
    movel([0.222983, -1.159035, -2.688254, -0.865100, 1.570796, 1.793779],accel_mss,speed_ms,0,blend_radius_m)
    movel([0.224864, -1.155909, -2.689612, -0.866867, 1.570796, 1.795661],accel_mss,speed_ms,0,blend_radius_m)
    movel([0.226758, -1.152767, -2.690968, -0.868654, 1.570796, 1.797554],accel_mss,speed_ms,0,blend_radius_m)
    movel([0.228663, -1.149608, -2.692321, -0.870460, 1.570796, 1.799459],accel_mss,speed_ms,0,blend_radius_m)
    movel([0.230579, -1.146433, -2.693671, -0.872285, 1.570796, 1.801376],accel_mss,speed_ms,0,blend_radius_m)
    movel([0.232508, -1.143242, -2.695017, -0.874130, 1.570796, 1.803304],accel_mss,speed_ms,0,blend_radius_m)
    movel([0.234448, -1.140034, -2.696360, -0.875995, 1.570796, 1.805244],accel_mss,speed_ms,0,blend_radius_m)
    movel([0.236400, -1.136809, -2.697701, -0.877879, 1.570796, 1.807197],accel_mss,speed_ms,0,blend_radius_m)
    movel([0.238365, -1.133567, -2.699038, -0.879784, 1.570796, 1.809161],accel_mss,speed_ms,0,blend_radius_m)
    speed_ms = 0.005
    # Splitting Linear movement in 6 (instruction 1650: MoveL 1560)
    movel([0.238365, -1.135190, -2.699886, -0.877313, 1.570796, 1.809161],accel_mss,speed_ms,0,blend_radius_m)
    movel([0.238365, -1.136822, -2.700732, -0.874835, 1.570796, 1.809161],accel_mss,speed_ms,0,blend_radius_m)
    movel([0.238365, -1.138461, -2.701578, -0.872351, 1.570796, 1.809161],accel_mss,speed_ms,0,blend_radius_m)
    movel([0.238365, -1.140107, -2.702421, -0.869860, 1.570796, 1.809161],accel_mss,speed_ms,0,blend_radius_m)
    movel([0.238365, -1.141762, -2.703264, -0.867363, 1.570796, 1.809161],accel_mss,speed_ms,0,blend_radius_m)
    movel([0.238365, -1.143424, -2.704104, -0.864860, 1.570796, 1.809161],accel_mss,speed_ms,0,blend_radius_m)
    speed_ms = 0.035
    movel([0.237244, -1.145248, -2.703344, -0.863797, 1.570796, 1.808041],accel_mss,speed_ms,0,blend_radius_m)
    movel([0.236530, -1.146827, -2.702683, -0.862879, 1.570796, 1.807326],accel_mss,speed_ms,0,blend_radius_m)
    movel([0.236456, -1.147482, -2.702408, -0.862499, 1.570796, 1.807252],accel_mss,speed_ms,0,blend_radius_m)
    movel([0.236644, -1.148017, -2.702183, -0.862189, 1.570796, 1.807440],accel_mss,speed_ms,0,blend_radius_m)
    movel([0.237148, -1.148420, -2.702014, -0.861955, 1.570796, 1.807944],accel_mss,speed_ms,0,blend_radius_m)
    movel([0.238856, -1.149021, -2.701761, -0.861607, 1.570796, 1.809652],accel_mss,speed_ms,0,blend_radius_m)
    movel([0.239312, -1.149732, -2.701461, -0.861196, 1.570796, 1.810108],accel_mss,speed_ms,0,blend_radius_m)
    movel([0.239253, -1.150736, -2.701036, -0.860617, 1.570796, 1.810049],accel_mss,speed_ms,0,blend_radius_m)
    movel([0.238982, -1.151334, -2.700783, -0.860272, 1.570796, 1.809779],accel_mss,speed_ms,0,blend_radius_m)
    movel([0.238533, -1.151984, -2.700507, -0.859898, 1.570796, 1.809329],accel_mss,speed_ms,0,blend_radius_m)
    movel([0.237724, -1.152770, -2.700173, -0.859446, 1.570796, 1.808520],accel_mss,speed_ms,0,blend_radius_m)
    movel([0.236706, -1.153477, -2.699872, -0.859040, 1.570796, 1.807503],accel_mss,speed_ms,0,blend_radius_m)
    movel([0.235633, -1.154037, -2.699633, -0.858718, 1.570796, 1.806429],accel_mss,speed_ms,0,blend_radius_m)
    movel([0.234658, -1.154376, -2.699489, -0.858524, 1.570796, 1.805454],accel_mss,speed_ms,0,blend_radius_m)
    movel([0.233282, -1.154589, -2.699397, -0.858402, 1.570796, 1.804078],accel_mss,speed_ms,0,blend_radius_m)
    movel([0.229282, -1.154746, -2.699331, -0.858313, 1.570796, 1.800079],accel_mss,speed_ms,0,blend_radius_m)
    movel([0.227820, -1.155045, -2.699203, -0.858141, 1.570796, 1.798617],accel_mss,speed_ms,0,blend_radius_m)
    movel([0.226445, -1.155548, -2.698987, -0.857853, 1.570796, 1.797242],accel_mss,speed_ms,0,blend_radius_m)
    movel([0.225160, -1.156247, -2.698688, -0.857454, 1.570796, 1.795956],accel_mss,speed_ms,0,blend_radius_m)
    movel([0.223977, -1.157137, -2.698306, -0.856946, 1.570796, 1.794773],accel_mss,speed_ms,0,blend_radius_m)
    movel([0.222904, -1.158203, -2.697847, -0.856339, 1.570796, 1.793700],accel_mss,speed_ms,0,blend_radius_m)
    movel([0.221945, -1.159439, -2.697314, -0.855636, 1.570796, 1.792742],accel_mss,speed_ms,0,blend_radius_m)
    movel([0.221112, -1.160835, -2.696709, -0.854844, 1.570796, 1.791908],accel_mss,speed_ms,0,blend_radius_m)
    movel([0.220408, -1.162386, -2.696036, -0.853967, 1.570796, 1.791204],accel_mss,speed_ms,0,blend_radius_m)
    movel([0.219938, -1.163796, -2.695421, -0.853172, 1.570796, 1.790734],accel_mss,speed_ms,0,blend_radius_m)
    movel([0.219697, -1.165056, -2.694871, -0.852463, 1.570796, 1.790493],accel_mss,speed_ms,0,blend_radius_m)
    movel([0.219689, -1.166162, -2.694385, -0.851842, 1.570796, 1.790485],accel_mss,speed_ms,0,blend_radius_m)
    movel([0.219908, -1.167132, -2.693959, -0.851298, 1.570796, 1.790705],accel_mss,speed_ms,0,blend_radius_m)
    movel([0.220362, -1.167961, -2.693594, -0.850834, 1.570796, 1.791158],accel_mss,speed_ms,0,blend_radius_m)
    movel([0.221050, -1.168660, -2.693286, -0.850444, 1.570796, 1.791847],accel_mss,speed_ms,0,blend_radius_m)
    movel([0.221971, -1.169234, -2.693032, -0.850123, 1.570796, 1.792768],accel_mss,speed_ms,0,blend_radius_m)
    movel([0.223127, -1.169689, -2.692831, -0.849870, 1.570796, 1.793923],accel_mss,speed_ms,0,blend_radius_m)
    movel([0.224501, -1.170243, -2.692585, -0.849561, 1.570796, 1.795298],accel_mss,speed_ms,0,blend_radius_m)
    movel([0.225596, -1.170958, -2.692268, -0.849163, 1.570796, 1.796392],accel_mss,speed_ms,0,blend_radius_m)
    movel([0.226416, -1.171837, -2.691877, -0.848675, 1.570796, 1.797212],accel_mss,speed_ms,0,blend_radius_m)
    movel([0.226961, -1.172885, -2.691410, -0.848094, 1.570796, 1.797757],accel_mss,speed_ms,0,blend_radius_m)
    movel([0.227234, -1.174102, -2.690867, -0.847420, 1.570796, 1.798030],accel_mss,speed_ms,0,blend_radius_m)
    movel([0.227236, -1.175490, -2.690245, -0.846655, 1.570796, 1.798032],accel_mss,speed_ms,0,blend_radius_m)
    movel([0.226973, -1.177048, -2.689544, -0.845797, 1.570796, 1.797769],accel_mss,speed_ms,0,blend_radius_m)
    movel([0.225772, -1.180845, -2.687826, -0.843718, 1.570796, 1.796568],accel_mss,speed_ms,0,blend_radius_m)
    movel([0.225687, -1.181482, -2.687536, -0.843370, 1.570796, 1.796483],accel_mss,speed_ms,0,blend_radius_m)
    movel([0.225807, -1.181899, -2.687347, -0.843143, 1.570796, 1.796603],accel_mss,speed_ms,0,blend_radius_m)
    movel([0.226148, -1.182136, -2.687239, -0.843014, 1.570796, 1.796944],accel_mss,speed_ms,0,blend_radius_m)
    movel([0.226739, -1.182219, -2.687201, -0.842969, 1.570796, 1.797536],accel_mss,speed_ms,0,blend_radius_m)
    movel([0.228756, -1.182074, -2.687267, -0.843048, 1.570796, 1.799553],accel_mss,speed_ms,0,blend_radius_m)
    movel([0.230313, -1.179268, -2.688542, -0.844579, 1.570796, 1.801110],accel_mss,speed_ms,0,blend_radius_m)
    movel([0.231361, -1.176537, -2.689774, -0.846078, 1.570796, 1.802157],accel_mss,speed_ms,0,blend_radius_m)
    movel([0.231901, -1.173941, -2.690939, -0.847509, 1.570796, 1.802697],accel_mss,speed_ms,0,blend_radius_m)
    movel([0.231933, -1.171540, -2.692009, -0.848840, 1.570796, 1.802729],accel_mss,speed_ms,0,blend_radius_m)
    movel([0.231460, -1.169398, -2.692959, -0.850032, 1.570796, 1.802256],accel_mss,speed_ms,0,blend_radius_m)
    movel([0.230481, -1.167579, -2.693762, -0.851048, 1.570796, 1.801277],accel_mss,speed_ms,0,blend_radius_m)
    movel([0.229004, -1.166141, -2.694394, -0.851853, 1.570796, 1.799801],accel_mss,speed_ms,0,blend_radius_m)
    movel([0.227028, -1.165156, -2.694826, -0.852406, 1.570796, 1.797824],accel_mss,speed_ms,0,blend_radius_m)
    movel([0.225461, -1.164723, -2.695016, -0.852650, 1.570796, 1.796257],accel_mss,speed_ms,0,blend_radius_m)
    movel([0.225184, -1.164402, -2.695157, -0.852831, 1.570796, 1.795980],accel_mss,speed_ms,0,blend_radius_m)
    movel([0.224965, -1.162873, -2.695824, -0.853692, 1.570796, 1.795761],accel_mss,speed_ms,0,blend_radius_m)
    movel([0.225058, -1.162007, -2.696201, -0.854181, 1.570796, 1.795855],accel_mss,speed_ms,0,blend_radius_m)
    movel([0.225320, -1.161132, -2.696581, -0.854676, 1.570796, 1.796116],accel_mss,speed_ms,0,blend_radius_m)
    movel([0.225746, -1.160709, -2.696764, -0.854916, 1.570796, 1.796542],accel_mss,speed_ms,0,blend_radius_m)
    movel([0.227523, -1.159789, -2.697163, -0.855438, 1.570796, 1.798319],accel_mss,speed_ms,0,blend_radius_m)
    movel([0.228367, -1.159533, -2.697273, -0.855583, 1.570796, 1.799163],accel_mss,speed_ms,0,blend_radius_m)
    movel([0.230926, -1.159334, -2.697359, -0.855696, 1.570796, 1.801723],accel_mss,speed_ms,0,blend_radius_m)
    movel([0.233469, -1.159205, -2.697415, -0.855769, 1.570796, 1.804265],accel_mss,speed_ms,0,blend_radius_m)
    movel([0.235371, -1.158792, -2.697593, -0.856004, 1.570796, 1.806168],accel_mss,speed_ms,0,blend_radius_m)
    movel([0.237250, -1.157990, -2.697939, -0.856460, 1.570796, 1.808047],accel_mss,speed_ms,0,blend_radius_m)
    movel([0.238179, -1.157418, -2.698185, -0.856786, 1.570796, 1.808975],accel_mss,speed_ms,0,blend_radius_m)
    movel([0.239098, -1.156716, -2.698487, -0.857186, 1.570796, 1.809894],accel_mss,speed_ms,0,blend_radius_m)
    movel([0.240913, -1.154875, -2.699275, -0.858239, 1.570796, 1.811709],accel_mss,speed_ms,0,blend_radius_m)
    movel([0.242527, -1.152630, -2.700233, -0.859527, 1.570796, 1.813323],accel_mss,speed_ms,0,blend_radius_m)
    movel([0.243579, -1.150494, -2.701139, -0.860757, 1.570796, 1.814376],accel_mss,speed_ms,0,blend_radius_m)
    movel([0.244075, -1.148524, -2.701970, -0.861895, 1.570796, 1.814872],accel_mss,speed_ms,0,blend_radius_m)
    movel([0.244018, -1.146789, -2.702699, -0.862901, 1.570796, 1.814815],accel_mss,speed_ms,0,blend_radius_m)
    movel([0.243413, -1.145345, -2.703304, -0.863741, 1.570796, 1.814209],accel_mss,speed_ms,0,blend_radius_m)
    movel([0.242264, -1.144262, -2.703756, -0.864371, 1.570796, 1.813060],accel_mss,speed_ms,0,blend_radius_m)
    movel([0.240580, -1.143600, -2.704031, -0.864757, 1.570796, 1.811376],accel_mss,speed_ms,0,blend_radius_m)
    movel([0.238365, -1.143424, -2.704104, -0.864860, 1.570796, 1.809161],accel_mss,speed_ms,0,blend_radius_m)
    movel([0.237244, -1.145248, -2.703344, -0.863797, 1.570796, 1.808041],accel_mss,speed_ms,0,blend_radius_m)
    movel([0.236549, -1.146782, -2.702702, -0.862905, 1.570796, 1.807346],accel_mss,speed_ms,0,blend_radius_m)
    speed_ms = 0.005
    # Splitting Linear movement in 20 (instruction 1731: MoveL 1639)
    movel([0.236549, -1.144293, -2.701444, -0.866652, 1.570796, 1.807346],accel_mss,speed_ms,0,blend_radius_m)
    movel([0.236549, -1.141822, -2.700183, -0.870385, 1.570796, 1.807346],accel_mss,speed_ms,0,blend_radius_m)
    movel([0.236549, -1.139368, -2.698918, -0.874103, 1.570796, 1.807346],accel_mss,speed_ms,0,blend_radius_m)
    movel([0.236549, -1.136931, -2.697650, -0.877808, 1.570796, 1.807346],accel_mss,speed_ms,0,blend_radius_m)
    movel([0.236549, -1.134512, -2.696379, -0.881499, 1.570796, 1.807346],accel_mss,speed_ms,0,blend_radius_m)
    movel([0.236549, -1.132109, -2.695104, -0.885175, 1.570796, 1.807346],accel_mss,speed_ms,0,blend_radius_m)
    movel([0.236549, -1.129724, -2.693827, -0.888838, 1.570796, 1.807346],accel_mss,speed_ms,0,blend_radius_m)
    movel([0.236549, -1.127356, -2.692546, -0.892487, 1.570796, 1.807346],accel_mss,speed_ms,0,blend_radius_m)
    movel([0.236549, -1.125005, -2.691262, -0.896122, 1.570796, 1.807346],accel_mss,speed_ms,0,blend_radius_m)
    movel([0.236549, -1.122671, -2.689975, -0.899743, 1.570796, 1.807346],accel_mss,speed_ms,0,blend_radius_m)
    movel([0.236549, -1.120354, -2.688684, -0.903351, 1.570796, 1.807346],accel_mss,speed_ms,0,blend_radius_m)
    movel([0.236549, -1.118053, -2.687391, -0.906945, 1.570796, 1.807346],accel_mss,speed_ms,0,blend_radius_m)
    movel([0.236549, -1.115769, -2.686095, -0.910526, 1.570796, 1.807346],accel_mss,speed_ms,0,blend_radius_m)
    movel([0.236549, -1.113501, -2.684795, -0.914093, 1.570796, 1.807346],accel_mss,speed_ms,0,blend_radius_m)
    movel([0.236549, -1.111250, -2.683493, -0.917647, 1.570796, 1.807346],accel_mss,speed_ms,0,blend_radius_m)
    movel([0.236549, -1.109015, -2.682187, -0.921187, 1.570796, 1.807346],accel_mss,speed_ms,0,blend_radius_m)
    movel([0.236549, -1.106796, -2.680878, -0.924714, 1.570796, 1.807346],accel_mss,speed_ms,0,blend_radius_m)
    movel([0.236549, -1.104594, -2.679567, -0.928228, 1.570796, 1.807346],accel_mss,speed_ms,0,blend_radius_m)
    movel([0.236549, -1.102407, -2.678252, -0.931729, 1.570796, 1.807346],accel_mss,speed_ms,0,blend_radius_m)
    movel([0.236549, -1.100237, -2.676935, -0.935217, 1.570796, 1.807346],accel_mss,speed_ms,0,blend_radius_m)
    speed_ms = 1.000
    movel([0.236549, -1.100237, -2.676935, -0.935217, 1.570796, 1.807346],accel_mss,speed_ms,0,blend_radius_m)
    # Splitting Linear movement in 30 (instruction 1734: MoveL 1641)
    movel([0.236549, -1.098082, -2.675615, -0.938692, 1.570796, 1.807346],accel_mss,speed_ms,0,blend_radius_m)
    movel([0.236549, -1.095943, -2.674292, -0.942154, 1.570796, 1.807346],accel_mss,speed_ms,0,blend_radius_m)
    movel([0.236549, -1.093820, -2.672966, -0.945603, 1.570796, 1.807346],accel_mss,speed_ms,0,blend_radius_m)
    movel([0.236549, -1.091713, -2.671637, -0.949039, 1.570796, 1.807346],accel_mss,speed_ms,0,blend_radius_m)
    movel([0.236549, -1.089621, -2.670305, -0.952463, 1.570796, 1.807346],accel_mss,speed_ms,0,blend_radius_m)
    movel([0.236549, -1.087545, -2.668970, -0.955874, 1.570796, 1.807346],accel_mss,speed_ms,0,blend_radius_m)
    movel([0.236549, -1.085484, -2.667633, -0.959272, 1.570796, 1.807346],accel_mss,speed_ms,0,blend_radius_m)
    movel([0.236549, -1.083438, -2.666293, -0.962658, 1.570796, 1.807346],accel_mss,speed_ms,0,blend_radius_m)
    movel([0.236549, -1.081407, -2.664950, -0.966031, 1.570796, 1.807346],accel_mss,speed_ms,0,blend_radius_m)
    movel([0.236549, -1.079392, -2.663605, -0.969392, 1.570796, 1.807346],accel_mss,speed_ms,0,blend_radius_m)
    movel([0.236549, -1.077392, -2.662256, -0.972741, 1.570796, 1.807346],accel_mss,speed_ms,0,blend_radius_m)
    movel([0.236549, -1.075406, -2.660905, -0.976077, 1.570796, 1.807346],accel_mss,speed_ms,0,blend_radius_m)
    movel([0.236549, -1.073436, -2.659552, -0.979402, 1.570796, 1.807346],accel_mss,speed_ms,0,blend_radius_m)
    movel([0.236549, -1.071480, -2.658195, -0.982714, 1.570796, 1.807346],accel_mss,speed_ms,0,blend_radius_m)
    movel([0.236549, -1.069539, -2.656837, -0.986014, 1.570796, 1.807346],accel_mss,speed_ms,0,blend_radius_m)
    movel([0.236549, -1.067612, -2.655475, -0.989302, 1.570796, 1.807346],accel_mss,speed_ms,0,blend_radius_m)
    movel([0.236549, -1.065701, -2.654111, -0.992578, 1.570796, 1.807346],accel_mss,speed_ms,0,blend_radius_m)
    movel([0.236549, -1.063803, -2.652744, -0.995842, 1.570796, 1.807346],accel_mss,speed_ms,0,blend_radius_m)
    movel([0.236549, -1.061920, -2.651375, -0.999094, 1.570796, 1.807346],accel_mss,speed_ms,0,blend_radius_m)
    movel([0.236549, -1.060051, -2.650003, -1.002335, 1.570796, 1.807346],accel_mss,speed_ms,0,blend_radius_m)
    movel([0.236549, -1.058197, -2.648629, -1.005564, 1.570796, 1.807346],accel_mss,speed_ms,0,blend_radius_m)
    movel([0.236549, -1.056356, -2.647252, -1.008781, 1.570796, 1.807346],accel_mss,speed_ms,0,blend_radius_m)
    movel([0.236549, -1.054530, -2.645872, -1.011987, 1.570796, 1.807346],accel_mss,speed_ms,0,blend_radius_m)
    movel([0.236549, -1.052717, -2.644491, -1.015181, 1.570796, 1.807346],accel_mss,speed_ms,0,blend_radius_m)
    movel([0.236549, -1.050918, -2.643106, -1.018364, 1.570796, 1.807346],accel_mss,speed_ms,0,blend_radius_m)
    movel([0.236549, -1.049134, -2.641719, -1.021536, 1.570796, 1.807346],accel_mss,speed_ms,0,blend_radius_m)
    movel([0.236549, -1.047363, -2.640330, -1.024696, 1.570796, 1.807346],accel_mss,speed_ms,0,blend_radius_m)
    movel([0.236549, -1.045605, -2.638939, -1.027845, 1.570796, 1.807346],accel_mss,speed_ms,0,blend_radius_m)
    movel([0.236549, -1.043861, -2.637545, -1.030983, 1.570796, 1.807346],accel_mss,speed_ms,0,blend_radius_m)
    movel([0.236549, -1.042131, -2.636148, -1.034110, 1.570796, 1.807346],accel_mss,speed_ms,0,blend_radius_m)
